(* CODESYS project BES3543.export

Project tree, tasks and I/O mapping:
  DATA_TYPE/
    data type EIXO_MOVER
    data type EIXO_STATUS
    data type RECEITA
    data type TURNOS_10
    function block COP [ST]
    function block FB_ATUADOR [ST]
    function block FB_Markem_SelecionarMacro [ST]
    function block FB_SMARTMOTOR [ST]
    program LEITURA_DATA_PLC [LD]
    function block RTON [FBD]
  D_PESAGEM/
    global variables GVL_PESAGEM
    program D00_PESAGEM [ST]
    program D01_EST_ETIQUETA [ST]
    program D02_SELEC_ETIQUETA [ST]
    program D03_ENTRADAS_REMOTAS [ST]
    program D04_SAIDAS_REMOTAS [ST]
  LADO_A/
    01 - LA_GERAL/
      global variables LA_GERAL
      program A00_ENTRADAS [ST]
      program A00_SAIDAS [ST]
      program A01_COMANDOS [ST]
      program A02_LAMPADAS [ST]
      program A03_COORDENADAS [ST]
      program ALARMES [ST]
    02 - LA_EMPILHADOR/
      global variables LA_EMP
      program B00_EMPILHA_SACOLA [ST]
      program B01_MANUAL [ST]
      program B02_EMPILHADOR_X [ST]
      program B03_INSPECAO [ST]
      program B04_ENTRADAS_REMOTAS [ST]
      program B05_SAIDAS_REMOTAS [ST]
    03 - LA_ENVOLVEDOR/
      global variables LA_ENV
      program C01_GIRO_SACOLA [ST]
      program C02_MANUAL [ST]
      program C03_EST_ENTRADA [ST]
      program C04_EST_TRANSPORTADOR [ST]
      program C05_EST_SAIDA [ST]
      program C06_ENTRADAS_REMOTAS [ST]
      program C07_SAIDAS_REMOTAS [ST]
    04 - LA_MOTION/
      program M0_LA_EMP_X [FBD]
      program M1_LA_EMP_GARRA [FBD]
      program M2_LA_EMP_GIRO [FBD]
      program M3_LA_ENV_Z [FBD]
      program M4_LA_ENV_X [FBD]
      program M5_LA_ENV_GIRO_LD [FBD]
      program M6_LA_ENV_GIRO_LE [FBD]
    05 - LA_IHM/
      global variables LA_IHM
      program E00_TELA_RECEITAS [ST]
      program E01_TELA_ATUADORES_EMPILHADOR [ST]
      program E02_TELA_ATUADORES_ENVOLVEDOR [ST]
      program E03_TELA_ATUADORES_PESAGEM [ST]
      program E04_TELA_OPERACAO [ST]
      program E05_CONTADORES [ST]
      program E06_HISTORICO [ST]
      program E07_HISTORICO_ESPELHAMENTO [ST]
  program TESTES_IOS [ST]
*)

// DATA_TYPE/EIXO_MOVER
TYPE EIXO_MOVER :
STRUCT
	
	sp_POSICAO			: LREAL;
	sp_VELOCIDADE		: LREAL;
	sp_ACELERACAO		: LREAL;
	sp_DESACELERACAO	: LREAL;

END_STRUCT
END_TYPE

// DATA_TYPE/EIXO_STATUS
TYPE EIXO_STATUS :
STRUCT
	
	bit_MOVE_FAZENDO		: BOOL;
	bit_MOVE_FEITO			: BOOL;
	bit_MOVE_ERRO			: BOOL;

END_STRUCT
END_TYPE

// DATA_TYPE/RECEITA
TYPE RECEITA :
STRUCT
	NOME 						: STRING;
	
	
//RECEITAS EMPILHADOR
	//CAMADAS MÁXIMAS DE EMPILHAMENTO / POSIÇÕES MÁXIMAS DE PEGA
	int_NUM_MAX_CAMADAS_EMPILHADOR	: INT;
	
	//CAMADA MÁXIMA DE EMPILHAMENTO ANTES DE ABAIXAR ATUADOR
	int_NUM_DESCER_MESA_EMPILHADOR	: INT;

	//GARRA EMPILHADOR
	coord_PRE_PEGA_GARRA_EMPILHADOR				: EIXO_MOVER;
	coord_PEGA_GARRA_EMPILHADOR					: EIXO_MOVER;
	
	sp_PRE_ENTREGA_GARRA_EMPILHADOR_POSICAO		: ARRAY[1..7] OF LREAL;
	sp_ENTREGA_GARRA_EMPILHADOR_VELOCIDADE		: LREAL;
	sp_ENTREGA_GARRA_EMPILHADOR_ACELERACAO		: LREAL;
	sp_ENTREGA_GARRA_EMPILHADOR_DESACELERACAO	: LREAL;
	
	sp_ENTREGA_GARRA_EMPILHADOR_POSICAO				: ARRAY[1..7] OF LREAL;
	sp_PRE_ENTREGA_GARRA_EMPILHADOR_VELOCIDADE		: LREAL;
	sp_PRE_ENTREGA_GARRA_EMPILHADOR_ACELERACAO		: LREAL;
	sp_PRE_ENTREGA_GARRA_EMPILHADOR_DESACELERACAO	: LREAL;
	
	tmr_TRANSICAO_ENTREGA_EMPILHADOR			: ARRAY[1..7] OF TIME;
	
	sp_POSICAO_ABRE_GARRA_EMPILHADOR			: ARRAY[1..7] OF LREAL;
	
	
	//EIXO X EMPILHADOR
	coord_X_EMPILHADOR_POS						: ARRAY[1..7] OF EIXO_MOVER;
	coord_X_EMPILHADOR_ENTREGA					: EIXO_MOVER;
	coord_X_EMPILHADOR_INSPECAO					: EIXO_MOVER;
	
	
	//MESA GIRO EMPILHADOR
	coord_MESA_GIRO_INICIAL				: EIXO_MOVER;
	coord_MESA_GIRO_FINAL				: EIXO_MOVER;
	coord_MESA_GIRO_INSPECAO			: EIXO_MOVER;
	
	
//RECEITAS ENVOLVEDOR
	//GIRO ENVOLVEDOR
	coord_GIRO_ENVOLVEDOR_PEGA			: EIXO_MOVER;
	coord_GIRO_ENVOLVEDOR_CORTE			: EIXO_MOVER;
	coord_GIRO_ENVOLVEDOR_ENTREGA		: EIXO_MOVER;
	
	//EIXO X ENVOLVEDOR
	coord_X_ENVOLVEDOR_PEGA				: EIXO_MOVER;
	coord_X_ENVOLVEDOR_CORTE			: EIXO_MOVER;
	coord_X_ENVOLVEDOR_ENTREGA			: EIXO_MOVER;
	
	//EIXO Z ENVOLVEDOR
	coord_Z_ENVOLVEDOR_PRE_PEGA			: EIXO_MOVER;
	coord_Z_ENVOLVEDOR_PEGA				: EIXO_MOVER;
	coord_Z_ENVOLVEDOR_SAIDA_PEGA		: EIXO_MOVER;
	coord_Z_ENVOLVEDOR_CORTE			: EIXO_MOVER;
	coord_Z_ENVOLVEDOR_ENTREGA			: EIXO_MOVER;
	
	int_NUMERO_GIROS_ENVOLVEDOR			: INT;
	
//PESO PILHA SACOLA
	num_PESO_SACOLA 				    : REAL;
			
END_STRUCT
END_TYPE

// DATA_TYPE/TURNOS_10
TYPE TURNOS_10 :
STRUCT
	PRIMEIRO		: ARRAY[0..9] OF DINT;
	SEGUNDO			: ARRAY[0..9] OF DINT;
	TERCEIRO		: ARRAY[0..9] OF DINT;
END_STRUCT
END_TYPE

// D_PESAGEM/GVL_PESAGEM
{attribute 'qualified_only'}
VAR_GLOBAL
	
	est_MESA_DE_TRANSFERENCIA				: BOOL;
	est_REJEITO_PRODUTO						: BOOL;
	est_TRANSPORTADOR_PESAGEM				: BOOL;
	est_TRANSPORTADOR_ESTAGIO_1				: BOOL;
	est_TRANNSPORTADOR_MERGER				: BOOL;
	
	est_MESA_DE_TRANSFERENCIA_REVERSE		: BOOL;
	est_TRANSPORTADOR_PESAGEM_REVERSE		: BOOL;
	
	
	bit_valv_ACIONAMENTO_TRANSFERENCIA		: BOOL;
	
	
	
	bit_PESANDO_PILHA_SACOLA				: BOOL;
	bit_ENVOLVEDOR_1						: BOOL;
	bit_ENVOLVEDOR_2						: BOOL;
	
	status_VALOR_PESAGEM					: WORD;
	array_ETIQUETA							: WORD;
	array_HIST_PESO							: WORD;
	
	
	bit_ENVOLVEDOR_ENVIANDO_PILHA_2			: BOOL;
	bit_PESAGEM_ATUAL						: BOOL;
	bit_PESAGEM_ERRO						: BOOL;
	bit_PESAGEM_OK							: BOOL;
	
	
//	ENTRADAS	============//============//============//============//============//============//============
	
	//E-16DIO - SLOT 5 (RMT50005)	
		di_SENS_MESA_TRANSFER_1				: BOOL;
		di_SENS_PRODUTO_BALANCA				: BOOL;
		di_BT_CMD1_INSPECAO_OK				: BOOL;
		di_feedback_ERRO_MESA_TRANSFER		: BOOL;
		di_feedback_ERRO_REJEITO_PRODUTO	: BOOL;
		di_SENS_MESA_TRANSFER_2				: BOOL;
		di_SENS_PRODUTO_REJEITO				: BOOL;
		di_SPEED_A_MERGER_1					: BOOL;
		
	//E-16DIO - SLOT 5 (RMT50006)	
		di_feedback_ERRO_ESTAGIO_1			: BOOL;
		di_SENS_TRANSFERENCIA_AV			: BOOL;
		di_SENS_ETIQUETADORA				: BOOL;
		di_SENS_POSICIONADOR_EMPILHADOR_RC	: BOOL;
		di_SENS_PRODUTO_DISPONIVEL			: BOOL;
		di_EST_MESA_TRANS_PESAGEM_DO1		: BOOL;
		di_SENS_TRANSFERENCIA_RC			: BOOL;
		di_SENS_PRODUTO_MERGER				: BOOL;
		di_SENS_POSICIONADOR_EMPILHADOR_AV	: BOOL;
		di_feedback_ERRO_MERGER_1			: BOOL;;
		
	
//	SAIDAS		============//============//============//============//============//============//============

	//E-16DIO - SLOT 5 (RMT50005)
		do_SPEED_A_MESA_TRANSFER		: BOOL;
		do_ATU_TRANSFERENCIA_RC			: BOOL;
		do_LAMP_INSPECAO_OK				: BOOL;
		do_REVERSE_MESA_TRANSFER		: BOOL;
		do_SPEED_B_MESA_TRANSFER		: BOOL;
		do_SPEED_A_REJEITO_PRODUTO		: BOOL;
		do_ATU_TRANSFERENCIA_AV			: BOOL;
		
	//E-16DIO - SLOT 6 (RMT50006)
		do_EST_MESA_TRANS_PESAGEM_DI2	: BOOL;
		do_EST_MESA_TRANS_PESAGEM_DI3	: BOOL;
		do_ATU_POSICIONADOR_RC			: BOOL;
		do_EST_MESA_TRANS_PESAGEM_DI1	: BOOL;
		do_SPEED_A_ESTAGIO_1			: BOOL;
		do_ATU_POSICIONADOR_AV			: BOOL;
		
	//E-16DIO - SLOT 7 (RMT50007)
		do_EST_BALANCA					: BOOL;
		do_est_BALANCA_REVERSE			: BOOL;
	
END_VAR

// LADO_A/01 - LA_GERAL/LA_GERAL
{attribute 'qualified_only'}
VAR_GLOBAL

//Teste teste teste	
//RECEITAS
	rec_IHM								: RECEITA;
	rec_SELECIONADA						: RECEITA;

//COMANDOS
	bit_MAQUINA_PRONTA				: BOOL;
	bit_MAQUINA_RODANDO				: BOOL;
	bit_MAQUINA_RESET				: BOOL;
	bit_MAQUINA_ESTAVEL				: BOOL;
	bit_SERVOS_RESET				: BOOL;
	bit_SAFETY_ATIVO				: BOOL;
	
	bit_MAQUINA_MANUAL				: BOOL;
	bit_BT_DESLIGA					: BOOL;
	
	
	bit_SERVOS_ENABLE				: BOOL;
	bit_AUTO_HABILITAR_EIXOS		: BOOL;
	bit_EIXO_X_EMPILHADOR_PRONTO	: BOOL;
	bit_EIXO_GARRA_EMPILHADOR_PRONTO : BOOL;
	bit_EIXO_GIRO_MESA_PRONTO		: BOOL;
	bit_EIXO_Z_ENVOLVEDOR_PRONTO	: BOOL;
	bit_EIXO_X_ENVOLVEDOR_PRONTO	: BOOL;
	bit_EIXO_GIRO_ENVOLVEDOR_LD_PRONTO : BOOL;
	bit_EIXO_GIRO_ENVOLVEDOR_LE_PRONTO : BOOL;
	bit_EIXOS_PRONTOS				: BOOL;
	
	TESTE_Z							: BOOL;
	RESET_Z							: BOOL;
	bit_TIRANDO_PRODUTO				: BOOL;
	bit_ALARME_SONORO_CASE			: BOOL;
	bit_SACOLA_POSICIONADA				: BOOL;
	tmr_CICLO_COMPLETO				: TON;

//LAMPADAS
	bit_LAMP_VERDE					: BOOL;
	bit_LAMP_VERMELHO				: BOOL;
	bit_LAMP_AMARELO				: BOOL;
	bit_LAMP_AZUL					: BOOL;
	bit_TL_SONORO					: BOOL;
	bit_LAMP_INSPECAO				: BOOL;
		
	bit_LAMP_VERDE_PULSO			: BOOL;
	bit_LAMP_VERMELHO_PULSO			: BOOL;
	bit_LAMP_AMARELO_PULSO			: BOOL;
	bit_LAMP_AZUL_PULSO				: BOOL;
	bit_TL_SONORO_PULSO				: BOOL;
	bit_LAMP_INSPECAO_PULSO			: BOOL;
	
//ALARMES
	status_alarm_EIXO_Y					: INT;
	status_alarm_EIXO_Z					: INT;
	status_alarm_EIXO_COLMEIA_1			: INT;
	status_alarm_EIXO_COLMEIA_2			: INT;
	status_alarm_atu_POSICIONA_PRODUTO	: INT;
	status_alarm_atu_STOP_ENTREGA		: INT;
	status_alarm_atu_STOP_PRE_ENTREGA	: INT;
	status_alarm_atu_MANI_GARRA			: INT;
	status_alarm_atu_PRODUTO_FREIO		: INT;
	status_alarm_atu_SEPARADOR_Y		: INT;
	status_alarm_atu_SEPARADOR_Z		: INT;
	status_alarm_atu_DIVERTER_FREIO		: INT;
	
	status_alarm_atu_FORM_PEGA_CAIXA	: INT;
	status_alarm_atu_FORM_FORMADOR		: INT;
	status_alarm_atu_FORM_EMPURADDOR	: INT;
	status_alarm_atu_FORM_VACUO			: INT;
	
	status_alarm_SAFETY_CASE			: INT;
	status_alarm_SAFETY_FORM			: INT;
	status_alarm_AR						: INT;
	
	status_alarm_in_PORTA_CASE_1		: INT;
	status_alarm_in_PORTA_CASE_2		: INT;
	status_alarm_in_PORTA_CASE_3		: INT;
	status_alarm_in_PORTA_CASE_4		: INT;
	status_alarm_in_PORTA_CASE_5		: INT;
	
	bit_STATUS_PARADA					: BOOL;
	bit_STATUS_OCIOSA					: BOOL;
	bit_STATUS_RODANDO					: BOOL;
	
	bit_TURNO_TROCADO					: BOOL;
	
	status_alarm_HOME_EIXO_Y			: INT;
	status_alarm_HOME_EIXO_Z			: INT;
	status_alarm_HOME_DIVERTER			: INT;
	status_alarm_ACUMULO_CAIXAS			: INT;
	status_alarm_in_PORTA_DIVERTER		: INT;
	status_alarm_VACUO_COLMEIA			: INT;
	status_alarm_NIVEL_COLMEIA			: INT;
	status_alarm_VACUO_PRODUTOS			: INT;
	status_alarm_INDEX_CAIXAS			: INT;
	status_alarm_COLMEIA_FREIO			: INT;
	status_alarm_BRACO_COLMEIA			: INT;
	status_alarm_FALTA_CAIXA			: INT;
	status_alarm_FALHA_PEGA				: INT;
	status_alarm_TEMP_COLA				: INT;
	status_alarm_NIVEL_COLA				: INT;
	status_alarm_BT_EMERGENCIA_CASE_1	: INT;
	status_alarm_BT_EMERGENCIA_CASE_2	: INT;
	status_alarm_BT_EMERGENCIA_FORM		: INT;
	atu_DESVIO_RODA						: BOOL;
	
	bit_ALARME_AR_CASE_ATIVO			: BOOL;
	bit_ALARME_FALTA_CAIXA_ATIVO		: BOOL;
	bit_SONORO_PULSO					: BOOL;
	
	r_trig_SEM_COLMEIA					: R_TRIG;
	r_trig_COLMEIA						: R_TRIG;
	bit_HABILITAR_EIXOS					: BOOL;
	
//	COORDENADAS	============//============//============//============//============//============//============
	
	//GARRA EMPILHADOR
	coord_GARRA_EMPILHADOR_PRE_PEGA						: EIXO_MOVER;
	coord_GARRA_EMPILHADOR_PEGA							: EIXO_MOVER;
	coord_GARRA_EMPILHADOR_PRE_ENTREGA					: EIXO_MOVER;
	coord_GARRA_EMPILHADOR_ENTREGA						: EIXO_MOVER;
	
	//EIXO X EMPILHADOR
	coord_X_EMPILHADOR_POS_1							: EIXO_MOVER;
	coord_X_EMPILHADOR_POS_2							: EIXO_MOVER;
	coord_X_EMPILHADOR_POS_3							: EIXO_MOVER;
	coord_X_EMPILHADOR_POS_4							: EIXO_MOVER;
	coord_X_EMPILHADOR_POS_5							: EIXO_MOVER;
	coord_X_EMPILHADOR_POS_6							: EIXO_MOVER;
	
	coord_X_EMPILHADOR_INSPECAO							: EIXO_MOVER;
	coord_X_EMPILHADOR_ENTREGA							: EIXO_MOVER;
	
	//MESA GIRO EMPILHADOR
	coord_MESA_GIRO_POSICAO_INICIAL						: EIXO_MOVER;
	coord_MESA_GIRO_POSICAO_FINAL						: EIXO_MOVER;
	coord_MESA_GIRO_POSICAO_INSPECAO					: EIXO_MOVER;
	
	
	//EIXO Z ENVOLVEDOR
	coord_Z_ENVOLVEDOR_PRE_PEGA							: EIXO_MOVER;
	coord_Z_ENVOLVEDOR_PEGA								: EIXO_MOVER;
	coord_Z_ENVOLVEDOR_SAIDA_PEGA						: EIXO_MOVER;
	coord_Z_ENVOLVEDOR_CORTE							: EIXO_MOVER;
	coord_Z_ENVOLVEDOR_ENTREGA							: EIXO_MOVER;
	
	
	//EIXO X ENVOLVEDOR
	coord_X_ENVOLVEDOR_PEGA								: EIXO_MOVER;
	coord_X_ENVOLVEDOR_CORTE							: EIXO_MOVER;
	coord_X_ENVOLVEDOR_ENTREGA							: EIXO_MOVER;
	
	
	//GIRO ENVOLVEDOR
	coord_GIRO_ENVOLVEDOR_PEGA							: EIXO_MOVER;
	coord_GIRO_ENVOLVEDOR_CORTE							: EIXO_MOVER;
	coord_GIRO_ENVOLVEDOR_ENTREGA						: EIXO_MOVER;
	
	
//	ENTRADAS	============//============//============//============//============//============//============

	//E-16DI - SLOT 1
		di_BT_CMD1_START				: BOOL;
		di_BT_CMD1_STOP					: BOOL;
		di_BT_CMD1_RESET				: BOOL;
		di_BT_CMD2_START				: BOOL;
		di_BT_CMD2_STOP					: BOOL;
		di_BT_CMD2_RESET				: BOOL;
		di_SEG_GERAL_ATIVA				: BOOL;
		di_SEG_INTERNA_ATIVA			: BOOL;
		di_SEG_PORTA_1					: BOOL;
		di_SEG_PORTA_2					: BOOL;
		
	//E-16DI - SLOT 2
		di_ENV_SENS_ATU_GARRA_LD_RC		: BOOL;
		di_ENV_SENS_ATU_GARRA_LE_RC		: BOOL;
		di_ENV_SENS_ATU_ABERTURA_AV		: BOOL;
		di_ENV_SENS_ATU_ABERTURA_RC		: BOOL;
	
//	SAIDAS		============//============//============//============//============//============//============

	//E-8DO - SLOT 3
		do_TL1_VERDE				: BOOL;
		do_TL1_VERMELHO				: BOOL;
		do_TL1_AMARELO				: BOOL;
		do_TL2_VERDE				: BOOL;
		do_TL2_VERMELHO				: BOOL;
		do_TL2_AMARELO				: BOOL;
		do_TL1_SONORO				: BOOL;
		do_SAIDA_COLAR_EQUIQUETA	: BOOL;
		
	//E-8DO - SLOT 4
		do_ENV_CORTE_FILME			: BOOL;
		
	//E-8DO - SLOT 5
		do_ENV_ATU_GARRAS			: BOOL;
		do_ENV_ATU_ABERTURA			: BOOL;	

	
	bit_MAQUINA_VAZIO					: BOOL;
	
	int_HIST_INDEX_TURNO1			: DINT;
	int_HIST_INDEX_TURNO2			: DINT;
	int_HIST_INDEX_TURNO3			: DINT;
	
	num_VOLTAS							: LREAL;
	
	bit_EIXO_GERAL_MOVENDO			: BOOL;
	
	bit_RESET_GERAL					: BOOL;
	
END_VAR

// LADO_A/02 - LA_EMPILHADOR/LA_EMP
{attribute 'qualified_only'}
VAR_GLOBAL
	
//COMANDOS

	bit_GARRA_EMPILHADOR_EXECUTANDO_RESET	: BOOL;
	bit_EIXO_X_EMPILHADOR_EXECUTANDO_RESET	: BOOL;
	bit_MESA_GIRO_EXECUTANDO_RESET			: BOOL;
	
	bit_ENTREGA_EMPILHADOR_CONCLUIDO		: BOOL;
	bit_ENTREGA_PILHA_CONCLUIDO				: BOOL;
	bit_EIXO_X_MOVE_CONCLUIDO				: BOOL;
	bit_MESA_GIRO_CONCLUIDO					: BOOL;
	
	bit_LIBERA_INSPECAO_PILHA				: BOOL;
	bit_EST_INSPECAO_ENTREGUE_1				: BOOL;
	bit_EST_INSPECAO_ENTREGUE_2				: BOOL;
	bit_OPERADOR_INSPECAO_OK				: BOOL;
	bit_EST_ENVIAR_PILHA_INSPECAO			: BOOL;
	bit_REALIZANDO_INSPECAO					: BOOL;
	
	bit_LIBERA_ENTREGA_PILHA				: BOOL;
	bit_ENTREGANDO_PILHA_COMPLETA			: BOOL;
	bit_EST_PILHA_ENTREGUE					: BOOL;
	
	bit_STATUS_INSPECAO_1					: BOOL;
	
	bit_LIBERA_PEGA							: BOOL;
	bit_LIBERA_GIRO							: BOOL;
	bit_LIBERA_X							: BOOL;
	
	bit_PILHA_PAR							: BOOL;
	bit_PILHA_IMPAR							: BOOL;
	
	bit_GIRO_MESA_REVERSE					: BOOL;
	bit_GIRO_MESA_FOWARD					: BOOL;
	
	bit_LIGA_EST_INSPECAO					: BOOL;
	bit_LIGA_EST_MESA_GIRO					: BOOL;
	
	
	bit_valv_GARRA_SACOLA					: BOOL;
	bit_valv_BANDEJA						: BOOL;
	bit_valv_DESCE_MESA_GIRO				: BOOL;
	bit_valv_POSICIONA_SACOLA				: BOOL;
	
	est_ROLETES_GIRO_MESA					: BOOL;
	est_INSPECAO_EMPILHADOR 				: BOOL;
	
	est_ROLETES_GIRO_MESA_REVERSE			: BOOL;
	est_INSPECAO_EMPILHADOR_REVERSE			: BOOL;
	
	
	
	
	bit_EIXO_X_EMPILHADOR_FAZER_HOME		: BOOL;
	bit_EIXO_X_EMPILHADOR_POSICIONADO		: BOOL;
	
	bit_EIXO_GIRO_MESA_FAZER_HOME			: BOOL;
	bit_EIXO_GIRO_MESA_POSICIONADO			: BOOL;
	
	bit_EIXO_GARRA_EMPILHADOR_FAZER_HOME	: BOOL;
	bit_EIXO_GARRA_EMPILHADOR_POSICIONADO	: BOOL;
	
	
	
	bit_EIXO_GARRA_EMPILHADOR_MOVER_ABS		: BOOL;
	bit_EIXO_GARRA_EMPILHADOR_MOVER_REL		: BOOL;
	
	bit_EIXO_X_EMPILHADOR_MOVER_ABS			: BOOL;
	bit_EIXO_X_EMPILHADOR_MOVER_REL			: BOOL;
	
	bit_EIXO_GIRO_MESA_MOVER_ABS			: BOOL;
	bit_EIXO_GIRO_MESA_MOVER_REL			: BOOL;
	

	
	bit_GARRA_EMPILHADOR_JOG_FORWARD		: BOOL;
	bit_GARRA_EMPILHADOR_JOG_REVERSE		: BOOL;
	bit_GARRA_EMPILHADOR_JOG_STOP			: BOOL;
	
	bit_EIXO_X_EMPILHADOR_JOG_FORWARD		: BOOL;
	bit_EIXO_X_EMPILHADOR_JOG_REVERSE		: BOOL;
	bit_EIXO_X_EMPILHADOR_JOG_STOP			: BOOL;
	
	bit_GIRO_MESA_JOG_FORWARD				: BOOL;
	bit_GIRO_MESA_JOG_REVERSE				: BOOL;
	bit_GIRO_MESA_JOG_STOP					: BOOL;
	
	
	info_MOTOR_GARRA_EMPILHADOR_POS_ATUAL	: LREAL;
	info_MOTOR_EIXO_X_EMPILHADOR_POS_ATUAL	: LREAL;
	info_MOTOR_GIRO_MESA_POS_ATUAL			: LREAL;
	
	
	num_GIROS_STRETCH					: LREAL;
	
	tmr_RTON_MOVE_1						: RTON;
	tmr_RTON_MOVE_2						: RTON;
	tmr_RTON_MOVE_3						: RTON;
	tmr_RTON_MOVE_4						: RTON;
	tmr_RTON_MOVE_5						: RTON;
	
	
	//	ENTRADAS	============//============//============//============//============//============//============
		
	//E-16DIO - SLOT 1 (RMT50001)	
		di_SENS_MESA_GIRO_RC				: BOOL;
		di_SENS_MESA_GIRO_MD				: BOOL;
		di_SENS_PINCA_GARRA_EMPILHADOR_RC	: BOOL;
		di_SENS_APOIO_BANDEJA_RC			: BOOL;
		di_SENS_EST_INSPEC_PRODUTO_1		: BOOL;
		di_SENS_MESA_GIRO_AV				: BOOL;
		di_SENS_PINCA_GARRA_EMPILHADOR_AV	: BOOL;
		di_SENS_APOIO_BANDEJA_AV			: BOOL;
		di_SENS_PRODUTO_MESA_GIRO			: BOOL;
		di_SENS_EST_INSPEC_PRODUTO_2		: BOOL;
		
	//E-16DIO - SLOT 2 (RMT50002)	
		di_feedback_ERRO_MESA_GIRO			: BOOL;
		di_feedback_ERRO_EST_INSPECAO		: BOOL;
		
	
	
//	SAIDAS		============//============//============//============//============//============//============

	//E-16DIO - SLOT 1 (RMT50001)		
		do_ATU_MESA_GIRO_RC				: BOOL;
		do_ATU_PINCA_GARRA_EMPILHADOR	: BOOL;
		do_ATU_MESA_GIRO_AV				: BOOL;
		do_ATU_BANDEJA_APOIO			: BOOL;
		
	//E-16DIO - SLOT 2 (RMT50002)	
		do_SPEED_A_MESA_GIRO			: BOOL;
		do_SPEED_A_EST_INSPECAO			: BOOL;
		do_REVERSE_MESA_GIRO			: BOOL;
		do_SPEED_B_MESA_GIRO			: BOOL;
		do_REVERSE_EST_INSPECAO			: BOOL;
		do_SPEED_B_EST_INSPECAO			: BOOL;
		
	
	
	
	
END_VAR

// LADO_A/03 - LA_ENVOLVEDOR/LA_ENV
{attribute 'qualified_only'}
VAR_GLOBAL

	//BITS DE COMANDOS
	bit_ENVOLVEDOR_SACOLA_POSICIONADA		: BOOL;
	bit_ENVOLVEDOR_SACOLA_DEPOSITANDO		: BOOL;
	bit_ENVOLVEDOR_SACOLA_DEPOSITADA		: BOOL;
	
	bit_ENVOLVEDOR_ENVIANDO_PILHA			: BOOL;
	
	
	bit_EST_ENTRADA_CHEIA					: BOOL;

	

	//ATUADORES
	bit_valv_APROX_GARRA			: BOOL;
	bit_valv_GARRA_DUPLA			: BOOL;
	bit_valv_CORTE_FILME			: BOOL;
	bit_valv_VACUO_FILME			: BOOL;
	bit_ENV_CORTE_FILME			: BOOL;
	bit_valv_FECHA_FILME_1			: BOOL;
	bit_valv_FECHA_FILME_2			: BOOL;
	bit_valv_FECHA_FILME_3			: BOOL;
	
	//ESTEIRAS
	est_ENTRADA_ENVOLVEDOR			: BOOL;
	est_TRANSPORTADOR_ENVOLVEDOR	: BOOL;
	est_SAIDA_ENVOLVEDOR			: BOOL;


	//BITS DE EIXOS
	bit_EIXO_Z_ENVOLVEDOR_FAZER_HOME			: BOOL;
	bit_EIXO_Z_ENVOLVEDOR_POSICIONADO			: BOOL;
	
	bit_EIXO_X_ENVOLVEDOR_FAZER_HOME			: BOOL;
	bit_EIXO_X_ENVOLVEDOR_POSICIONADO			: BOOL;

	bit_EIXO_GIRO_ENVOLVEDOR_LD_FAZER_HOME		: BOOL;
	bit_EIXO_GIRO_ENVOLVEDOR_LD_POSICIONADO		: BOOL;
	
	bit_EIXO_GIRO_ENVOLVEDOR_LE_FAZER_HOME		: BOOL;
	bit_EIXO_GIRO_ENVOLVEDOR_LE_POSICIONADO		: BOOL;
	
	
	
	bit_EIXO_Z_ENVOLVEDOR_MOVER_ABS				: BOOL;
	bit_EIXO_Z_ENVOLVEDOR_MOVER_REL				: BOOL;
	
	bit_EIXO_X_ENVOLVEDOR_MOVER_ABS				: BOOL;
	bit_EIXO_X_ENVOLVEDOR_MOVER_REL				: BOOL;
	
	bit_EIXO_GIRO_ENVOLVEDOR_LD_MOVER_ABS		: BOOL;
	bit_EIXO_GIRO_ENVOLVEDOR_LD_MOVER_REL		: BOOL;
	
	bit_EIXO_GIRO_ENVOLVEDOR_LE_MOVER_ABS		: BOOL;
	bit_EIXO_GIRO_ENVOLVEDOR_LE_MOVER_REL		: BOOL;
	
	
	bit_MOTOR_Z_ENVOLVEDOR_JOG_FORWARD			: BOOL;
	bit_MOTOR_Z_ENVOLVEDOR_JOG_REVERSE			: BOOL;
	bit_MOTOR_Z_ENVOLVEDOR_JOG_STOP				: BOOL;
	
	bit_MOTOR_X_ENVOLVEDOR_JOG_FORWARD			: BOOL;
	bit_MOTOR_X_ENVOLVEDOR_JOG_REVERSE			: BOOL;
	bit_MOTOR_X_ENVOLVEDOR_JOG_STOP				: BOOL;
	
	bit_MOTOR_GIRO_ENVOLVEDOR_LD_JOG_FORWARD	: BOOL;
	bit_MOTOR_GIRO_ENVOLVEDOR_LD_JOG_REVERSE	: BOOL;
	bit_MOTOR_GIRO_ENVOLVEDOR_LD_JOG_STOP		: BOOL;
	
	bit_MOTOR_GIRO_ENVOLVEDOR_LE_JOG_FORWARD	: BOOL;
	bit_MOTOR_GIRO_ENVOLVEDOR_LE_JOG_REVERSE	: BOOL;
	bit_MOTOR_GIRO_ENVOLVEDOR_LE_JOG_STOP		: BOOL;
	
	info_MOTOR_GIRO_ENVOLVIMENTO_LD_POS_ATUAL	: LREAL;
	info_MOTOR_GIRO_ENVOLVIMENTO_LE_POS_ATUAL	: LREAL;
	
	info_MOTOR_Z_ENVOLVEDOR_POS_ATUAL			: LREAL;
	info_MOTOR_X_ENVOLVEDOR_POS_ATUAL			: LREAL;

	
	
//	ENTRADAS	============//============//============//============//============//============//============

	
	//E-16DIO - SLOT 3 (RMT50003)	
		di_SENS_EST_TRANS_PRESENCA			: BOOL;
		di_SENS_POS_2_ENVOLVEDOR			: BOOL;
		di_SENS_CORTE_FILME_RC				: BOOL;
		di_feedback_ERRO_ENTRADA_ENVOLVEDOR : BOOL;
		di_SENS_POS_1_ENVOLVEDOR			: BOOL;
		di_SENS_FILME_ENVOLVEDOR			: BOOL;
		di_SENS_CORTE_FILME_AV				: BOOL;
	
	//E-16DIO - SLOT 4 (RMT50004)		
		di_SENS_SAIDA_ENVOLVEDOR_1			: BOOL;
		di_SENS_SAIDA_ENVOLVEDOR_3			: BOOL;
		di_SENS_FECHA_FILME_1_RC			: BOOL;
		di_SENS_FECHA_FILME_2_RC			: BOOL;
		di_SENS_FECHA_FILME_3_RC			: BOOL;
		di_feedback_ERRO_TRANSP_SAIDA_1		: BOOL;
		di_SENS_SAIDA_ENVOLVEDOR_2			: BOOL;
		di_SENS_SAIDA_ENVOLVEDOR_4			: BOOL;
		di_SENS_FECHA_FILME_2_AV			: BOOL;
		di_SENS_FECHA_FILME_3_AV			: BOOL;

		
		
//	SAIDAS		============//============//============//============//============//============//============

	//E-16DIO - SLOT 3 (RMT50003)	
		do_EST_TRANS_ENVOLVEDOR_DI2		: BOOL;
		do_EST_TRANS_ENVOLVEDOR_DI3		: BOOL;
		do_VALV_CORTE_FILME				: BOOL;
		do_SPEED_A_ENTRADA_ENVOLVEDOR	: BOOL;
		do_EST_TRANS_ENVOLVEDOR_DI1		: BOOL;
		do_EST_TRANS_ENVOLVEDOR_DO1		: BOOL;
		do_VALV_VACUO_FILME				: BOOL;
		
	//E-16DIO - SLOT 4 (RMT50004)
		do_VALV_FECHA_FILME_2			: BOOL;
		do_SPEED_A_TRANSP_SAIDA_1		: BOOL;
		do_VALV_FECHA_FILME_1			: BOOL;
		do_VALV_FECHA_FILME_3			: BOOL;
	
	
END_VAR

// LADO_A/05 - LA_IHM/LA_IHM
{attribute 'qualified_only'}
VAR_GLOBAL
	
//Tela de Operação
	bit_MAQUINA_MANUAL				: BOOL;
	bit_MANUAL_HABILITAR_EIXOS		: BOOL;
	bit_bt_INSPECAO_OK				: BOOL;
	bit_STATUS_INSPECAO_OK			: INT;
	bit_STATUS_PESAGEM				: INT;
	
	
	array_HIST_ERRO_PESAGEM_1		: BOOL;
	array_HIST_ERRO_PESAGEM_2		: BOOL;
	array_HIST_ERRO_PESAGEM_3		: BOOL;
	array_HIST_ERRO_PESAGEM_4		: BOOL;
	array_HIST_ERRO_PESAGEM_5		: BOOL;
	array_HIST_ERRO_PESAGEM_6		: BOOL;
	array_HIST_ERRO_PESAGEM_7		: BOOL;


//ICONES DE ALARME NOS EIXOS
	bit_EIXO_X_EMPILHADOR_ALARME_ATIVO			: BOOL;
	bit_EIXO_GARRA_EMPILHADOR_ALARME_ATIVO		: BOOL;
	bit_EIXO_GIRO_MESA_ALARME_ATIVO				: BOOL;
	bit_EIXO_Z_ENVOLVEDOR_ALARME_ATIVO			: BOOL;
	bit_EIXO_X_ENVOLVEDOR_ALARME_ATIVO			: BOOL;
	bit_EIXO_GIRO_ENVOLVEDOR_LD_ALARME_ATIVO	: BOOL;
	bit_EIXO_GIRO_ENVOLVEDOR_LE_ALARME_ATIVO	: BOOL;
	bit_EIXO_GERAL_SAFETY						: BOOL;

//ICONES DE EIXOS HABILITADOS	
	bit_EIXO_X_EMPILHADOR_HABILITADO			: BOOL;
	bit_EIXO_GARRA_EMPILHADOR_HABILITADO		: BOOL;
	bit_EIXO_GIRO_MESA_HABILITADO				: BOOL;
	bit_EIXO_Z_ENVOLVEDOR_HABILITADO			: BOOL;
	bit_EIXO_X_ENVOLVEDOR_HABILITADO			: BOOL;
	bit_EIXO_GIRO_ENVOLVEDOR_LD_HABILITADO		: BOOL;
	bit_EIXO_GIRO_ENVOLVEDOR_LE_HABILITADO		: BOOL;
	
//ICONES PARA MOVIMENTOS JOG DOS EIXOS	
	bit_EIXO_X_EMPILHADOR_JOG_POSITIVO			: BOOL;
	bit_EIXO_X_EMPILHADOR_JOG_NEGATIVO			: BOOL;
	bit_EIXO_GARRA_EMPILHADOR_JOG_POSITIVO		: BOOL;
	bit_EIXO_GARRA_EMPILHADOR_JOG_NEGATIVO		: BOOL;
	bit_EIXO_GIRO_MESA_JOG_POSITIVO				: BOOL;
	bit_EIXO_GIRO_MESA_JOG_NEGATIVO				: BOOL;
	bit_EIXO_Z_ENVOLVEDOR_JOG_POSITIVO			: BOOL;
	bit_EIXO_Z_ENVOLVEDOR_JOG_NEGATIVO			: BOOL;
	bit_EIXO_X_ENVOLVEDOR_JOG_POSITIVO			: BOOL;
	bit_EIXO_X_ENVOLVEDOR_JOG_NEGATIVO			: BOOL;
	bit_EIXO_GIRO_ENVOLVEDOR_LD_JOG_POSITIVO	: BOOL;
	bit_EIXO_GIRO_ENVOLVEDOR_LD_JOG_NEGATIVO	: BOOL;
	bit_EIXO_GIRO_ENVOLVEDOR_LE_JOG_POSITIVO	: BOOL;
	bit_EIXO_GIRO_ENVOLVEDOR_LE_JOG_NEGATIVO	: BOOL;
	
//ICONES PARA FAZER HOME DOS EIXOS	
	bit_EIXO_X_EMPILHADOR_FAZER_HOME			: BOOL;
	bit_EIXO_GARRA_EMPILHADOR_FAZER_HOME		: BOOL;
	bit_EIXO_GIRO_MESA_FAZER_HOME				: BOOL;
	bit_EIXO_Z_ENVOLVEDOR_FAZER_HOME			: BOOL;
	bit_EIXO_X_ENVOLVEDOR_FAZER_HOME			: BOOL;
	bit_EIXO_GIRO_ENVOLVEDOR_LD_FAZER_HOME		: BOOL;
	bit_EIXO_GIRO_ENVOLVEDOR_LE_FAZER_HOME		: BOOL;
	
	
	//ICONES DE STATUS DO HOME DOS EIXOS
	bit_EIXO_X_EMPILHADOR_FAZENDO_HOME			: BOOL;
	bit_EIXO_GARRA_EMPILHADOR_FAZENDO_HOME		: BOOL;
	bit_EIXO_GIRO_MESA_FAZENDO_HOME				: BOOL;
	bit_EIXO_Z_ENVOLVEDOR_FAZENDO_HOME			: BOOL;
	bit_EIXO_X_ENVOLVEDOR_FAZENDO_HOME			: BOOL;
	bit_EIXO_GIRO_ENVOLVEDOR_LD_FAZENDO_HOME	: BOOL;
	bit_EIXO_GIRO_ENVOLVEDOR_LE_FAZENDO_HOME	: BOOL;
	
		
//INFORMAÇÃO DE POSIÇÃO ATUAL
	info_MANI_POS_ATUAL_X_EMPILHADOR			: LREAL;
	info_MANI_POS_ATUAL_GIRO_MESA				: LREAL;
	info_MANI_POS_ATUAL_Z_ENVOLVEDOR			: LREAL;
	info_MANI_POS_ATUAL_X_ENVOLVEDOR			: LREAL;
	info_MANI_POS_ATUAL_GARRA_EMPILHADOR		: LREAL;
	info_POS_ATUAL_GIRO_EMPILHADOR_LD			: LREAL;
	info_POS_ATUAL_GIRO_EMPILHADOR_LE			: LREAL;
	
	
//ICONES DE ALARME NOS MOTORES
	bit_feedback_ERRO_MESA_GIRO				: BOOL;
	bit_feedback_ERRO_EST_INSPECAO			: BOOL;
	bit_feedback_ERRO_ENTRADA_ENVOLVEDOR	: BOOL;
	bit_feedback_ERRO_TRANSP_SAIDA_1		: BOOL;
	bit_feedback_ERRO_MESA_TRANSFER			: BOOL;
	bit_feedback_ERRO_REJEITO_PRODUTO		: BOOL;
	bit_feedback_ERRO_ESTAGIO_1				: BOOL;
	bit_feedback_ERRO_MERGER_1				: BOOL;
	
	
	
	bit_GIRO_SACOLA_RESET			: BOOL;
	bit_GIRO_EMPILHAMENTO_RESET		: BOOL;
	
	sp_MANI_VELOCIDADE				: UINT;
	
	int_CAMADA_ATUAL				: INT	:=	1;
	
	bit_SIMULA_PEGA					: BOOL;
	bit_SIMULA_GIRO					: BOOL;
	bit_bt_RESET_SERVO				: BOOL;

// Tela de Receita
	bt_CARREGAR_RECEITA				: BOOL;
	bt_SALVAR_RECEITA				: BOOL;
	bt_UPLOAD_RECEITA				: BOOL;
	bt_DOWNLOAD_RECEITA				: BOOL;
	
	int_RECEITA_ATUAL				: INT;
	int_STATUS_RECEITA				: INT;
	
	
	bit_SELEC_RECEITA_1				: BOOL;
	bit_SELEC_RECEITA_2				: BOOL;
	bit_SELEC_RECEITA_3				: BOOL;
	bit_SELEC_RECEITA_4				: BOOL;
	bit_SELEC_RECEITA_5				: BOOL;
	bit_SELEC_RECEITA_6				: BOOL;
	bit_SELEC_RECEITA_7				: BOOL;
	bit_SELEC_RECEITA_8				: BOOL;
	bit_SELEC_RECEITA_9				: BOOL;
	bit_SELEC_RECEITA_10			: BOOL;
	
	
	nome_RECEITA_1							: STRING;
	nome_RECEITA_2							: STRING;
	nome_RECEITA_3							: STRING;
	nome_RECEITA_4							: STRING;
	nome_RECEITA_5							: STRING;
	nome_RECEITA_6							: STRING;
	nome_RECEITA_7							: STRING;
	nome_RECEITA_8							: STRING;
	nome_RECEITA_9							: STRING;
	nome_RECEITA_10							: STRING;
	
	
	ALARME_ATIVO					: BOOL;
	
	TEMPO_1				: TIME;
	TEMPO_2				: TIME;
	TEMPO_3				: TIME;
	TEMPO_4				: TIME;
	TEMPO_5				: TIME;
	TEMPO_TOTAL			: TIME;
	TEMPO_TOTAL_2		: TIME;
	
	bit_RESET_RTON		: BOOL;
	
//CONTADORES DE TEMPO DE MAQUINA
	//TURNO 1
	num_MAQUINA_RODANDO_SEGUNDOS_T1	: DINT;
	num_MAQUINA_RODANDO_MINUTOS_T1	: DINT;
	num_MAQUINA_RODANDO_HORAS_T1	: DINT;
	
	num_MAQUINA_PARADA_SEGUNDOS_T1	: DINT;
	num_MAQUINA_PARADA_MINUTOS_T1	: DINT;
	num_MAQUINA_PARADA_HORAS_T1		: DINT;
	
	num_MAQUINA_OCIOSA_SEGUNDOS_T1	: DINT;
	num_MAQUINA_OCIOSA_MINUTOS_T1	: DINT;
	num_MAQUINA_OCIOSA_HORAS_T1		: DINT;
	
	
	//TURNO 2
	num_MAQUINA_RODANDO_SEGUNDOS_T2	: DINT;
	num_MAQUINA_RODANDO_MINUTOS_T2	: DINT;
	num_MAQUINA_RODANDO_HORAS_T2	: DINT;
	
	num_MAQUINA_PARADA_SEGUNDOS_T2	: DINT;
	num_MAQUINA_PARADA_MINUTOS_T2	: DINT;
	num_MAQUINA_PARADA_HORAS_T2		: DINT;
	
	num_MAQUINA_OCIOSA_SEGUNDOS_T2	: DINT;
	num_MAQUINA_OCIOSA_MINUTOS_T2	: DINT;
	num_MAQUINA_OCIOSA_HORAS_T2		: DINT;
	
	
	//TURNO 3
	num_MAQUINA_RODANDO_SEGUNDOS_T3	: DINT;
	num_MAQUINA_RODANDO_MINUTOS_T3	: DINT;
	num_MAQUINA_RODANDO_HORAS_T3	: DINT;
	
	num_MAQUINA_PARADA_SEGUNDOS_T3	: DINT;
	num_MAQUINA_PARADA_MINUTOS_T3	: DINT;
	num_MAQUINA_PARADA_HORAS_T3		: DINT;
	
	num_MAQUINA_OCIOSA_SEGUNDOS_T3	: DINT;
	num_MAQUINA_OCIOSA_MINUTOS_T3	: DINT;
	num_MAQUINA_OCIOSA_HORAS_T3		: DINT;
	
	
	//CONTADORES
	time_SEGUNDOS					: INT;
	time_MINUTOS					: INT;
	time_HORAS						: INT;
	time_DIA						: INT;
	time_MES						: INT;
	time_ANO						: INT;
	
	bit_HORARIO_MINUTO_COMPLETO		: BOOL;
	bit_HORARIO_HORA_COMPLETO		: BOOL;
	bit_HORARIO_DIA_COMPLETO		: BOOL;
	bit_HORARIO_DIA_COMPLETO_REAL	: BOOL;
	bit_CONTADORES_RESET			: BOOL;
	
	num_PILHAS_COMPLETADAS_T1		: LREAL;
	num_PILHAS_COMPLETADAS_T2		: LREAL;
	num_PILHAS_COMPLETADAS_T3		: LREAL;
	
	num_PILHAS_REJEITADAS_T1		: LREAL;
	num_PILHAS_REJEITADAS_T2		: LREAL;
	num_PILHAS_REJEITADAS_T3		: LREAL;
	
	num_PILHAS_TOTAL_T1				: LREAL;
	num_PILHAS_TOTAL_T2				: LREAL;
	num_PILHAS_TOTAL_T3				: LREAL;

	
	tmr_MAQUINA_RODANDO_T1			: DINT;
	tmr_MAQUINA_RODANDO_T2			: DINT;
	tmr_MAQUINA_RODANDO_T3			: DINT;
	
	tmr_MAQUINA_PARADA_T1			: DINT;
	tmr_MAQUINA_PARADA_T2			: DINT;
	tmr_MAQUINA_PARADA_T3			: DINT;
	
	tmr_MAQUINA_OCIOSA_T1			: DINT;
	tmr_MAQUINA_OCIOSA_T2			: DINT;
	tmr_MAQUINA_OCIOSA_T3			: DINT;
	
	
	num_PORCENTAGEM_COMPLETADAS_T1 			: REAL;
	num_PORCENTAGEM_COMPLETADAS_T2 			: REAL;
	num_PORCENTAGEM_COMPLETADAS_T3 			: REAL;
	num_PORCENTAGEM_REJEITADAS_T1			: REAL;
	num_PORCENTAGEM_REJEITADAS_T2 			: REAL;
	num_PORCENTAGEM_REJEITADAS_T3 			: REAL;
	
	ihm_HIST_PORCENTAGEM_COMPLETADAS_T1		: DINT;
	ihm_HIST_PORCENTAGEM_COMPLETADAS_T2		: DINT;
	ihm_HIST_PORCENTAGEM_COMPLETADAS_T3		: DINT;
	ihm_HIST_PORCENTAGEM_REJEITADAS_T1		: DINT;
	ihm_HIST_PORCENTAGEM_REJEITADAS_T2		: DINT;
	ihm_HIST_PORCENTAGEM_REJEITADAS_T3		: DINT;
	
	
	info_DIA_ANTERIOR				: DINT;
	info_MES_ANTERIOR				: DINT;
	
	turno_A							: BOOL;
	turno_B							: BOOL;
	turno_C							: BOOL;
	
	ihm_HIST_INDEX_TURNO1			: ARRAY[0..9] OF BOOL;
	ihm_HIST_INDEX_TURNO2			: ARRAY[0..9] OF BOOL;
	ihm_HIST_INDEX_TURNO3			: ARRAY[0..9] OF BOOL;
	
	
	
	ONS_DIA_COMPLETO_1				: R_TRIG;;
	
	
//COP DIA 1
	COP_ihm_DIA_TURNO				: COP;
	COP_ihm_DIA_TURNO_AUX			: COP;
	
	COP_ihm_MES_TURNO				: COP;
	COP_ihm_MES_TURNO_AUX			: COP;
	
	COP_ihm_RODANDO_TURNO			: COP;
	COP_ihm_RODANDO_TURNO_AUX		: COP;
	
	COP_ihm_PARADO_TURNO			: COP;
	COP_ihm_PARADO_TURNO_AUX		: COP;
	
	COP_ihm_OCIOSO_TURNO			: COP;
	COP_ihm_OCIOSO_TURNO_AUX		: COP;

	COP_ihm_PILHAS_COMPLETADAS_TURNO		: COP;
	COP_ihm_PILHAS_COMPLETADAS_TURNO_AUX	: COP;	
	
	COP_ihm_PILHAS_REJEITADAS_TURNO			: COP;
	COP_ihm_PILHAS_REJEITADAS_TURNO_AUX		: COP;	
	
	COP_ihm_PILHAS_TOTAL_TURNO				: COP;
	COP_ihm_PILHAS_TOTAL_TURNO_AUX			: COP;	

	
	COP_ihm_PORCENTAGEM_COMPLETADAS			: COP;
	COP_ihm_PORCENTAGEM_COMPLETADAS_AUX		: COP;
	
	COP_ihm_PORCENTAGEM_REJEITADAS			: COP;
	COP_ihm_PORCENTAGEM_REJEITADAS_AUX		: COP;
	
	
//COP DIA 2
	COP_ihm_DIA_TURNO2				: COP;
	COP_ihm_DIA_TURNO_AUX2			: COP;
	
	COP_ihm_MES_TURNO2				: COP;
	COP_ihm_MES_TURNO_AUX2			: COP;
	
	COP_ihm_RODANDO_TURNO2			: COP;
	COP_ihm_RODANDO_TURNO_AUX2		: COP;
	
	COP_ihm_PARADO_TURNO2			: COP;
	COP_ihm_PARADO_TURNO_AUX2		: COP;
	
	COP_ihm_OCIOSO_TURNO2			: COP;
	COP_ihm_OCIOSO_TURNO_AUX2		: COP;

	COP_ihm_PILHAS_COMPLETADAS_TURNO2		: COP;
	COP_ihm_PILHAS_COMPLETADAS_TURNO_AUX2	: COP;	
	
	COP_ihm_PILHAS_REJEITADAS_TURNO2		: COP;
	COP_ihm_PILHAS_REJEITADAS_TURNO_AUX2	: COP;	
	
	COP_ihm_PILHAS_TOTAL_TURNO2				: COP;
	COP_ihm_PILHAS_TOTAL_TURNO_AUX2			: COP;	

	
	COP_ihm_PORCENTAGEM_COMPLETADAS2		: COP;
	COP_ihm_PORCENTAGEM_COMPLETADAS_AUX2	: COP;
	
	COP_ihm_PORCENTAGEM_REJEITADAS2			: COP;
	COP_ihm_PORCENTAGEM_REJEITADAS_AUX2		: COP;
	
	
//COP DIA 3
	COP_ihm_DIA_TURNO3				: COP;
	COP_ihm_DIA_TURNO_AUX3			: COP;
	
	COP_ihm_MES_TURNO3				: COP;
	COP_ihm_MES_TURNO_AUX3			: COP;
	
	COP_ihm_RODANDO_TURNO3			: COP;
	COP_ihm_RODANDO_TURNO_AUX3		: COP;
	
	COP_ihm_PARADO_TURNO3			: COP;
	COP_ihm_PARADO_TURNO_AUX3		: COP;
	
	COP_ihm_OCIOSO_TURNO3			: COP;
	COP_ihm_OCIOSO_TURNO_AUX3		: COP;

	COP_ihm_PILHAS_COMPLETADAS_TURNO3		: COP;
	COP_ihm_PILHAS_COMPLETADAS_TURNO_AUX3	: COP;	
	
	COP_ihm_PILHAS_REJEITADAS_TURNO3		: COP;
	COP_ihm_PILHAS_REJEITADAS_TURNO_AUX3	: COP;	
	
	COP_ihm_PILHAS_TOTAL_TURNO3				: COP;
	COP_ihm_PILHAS_TOTAL_TURNO_AUX3			: COP;	

	
	COP_ihm_PORCENTAGEM_COMPLETADAS3		: COP;
	COP_ihm_PORCENTAGEM_COMPLETADAS_AUX3	: COP;
	
	COP_ihm_PORCENTAGEM_REJEITADAS3			: COP;
	COP_ihm_PORCENTAGEM_REJEITADAS_AUX3		: COP;
	
	
	HORARIO_ATUAL_ANO				: YEAR;
	HORARIO_ATUAL_MES				: MONTH;
	HORARIO_ATUAL_DIA				: DAY;
	HORARIO_ATUAL_HORA				: HOUR;
	HORARIO_ATUAL_MINUTO			: MINUTE;
	HORARIO_ATUAL_SEGUNDO			: SECOND;
	
//BITS ATUADORES MODO MANUAL

	//ESTEIRAS DO EMPILHAMENTO DE SACOLA
	est_ROLETES_GIRO_MESA					: BOOL;
	est_INSPECAO_EMPILHADOR 				: BOOL;
	est_ROLETES_GIRO_MESA_REVERSE			: BOOL;
	est_INSPECAO_EMPILHADOR_REVERSE			: BOOL;

	//ESTEIRAS DO ENVOLVEDOR
	est_ENVOLVEDOR_ENTRADA					: BOOL;
	est_TRANSPORTADOR_ENVOLVEDOR			: BOOL;
	est_ENVOLVEDOR_SAIDA					: BOOL;
	
	//ESTEIRAS PARA REALIZAR PESAGEM DE SACOLAS
	est_MESA_DE_TRANSFERENCIA				: BOOL;
	est_REJEITO_PRODUTO						: BOOL;
	est_TRANSPORTADOR_PESAGEM				: BOOL;
	est_TRANSPORTADOR_ESTAGIO_1				: BOOL;
	est_TRANNSPORTADOR_MERGER				: BOOL;
	est_MESA_DE_TRANSFERENCIA_REVERSE		: BOOL;
	est_TRANSPORTADOR_PESAGEM_REVERSE		: BOOL;
	
	//BITS DE SELEÇÃO DE ATUADOR
	int_EMPILHADOR_ATUADOR_SELECIONADO		: INT;
	int_ENVOLVEDOR_ATUADOR_SELECIONADO		: INT;
	int_PESAGEM_ATUADOR_SELECIONADO			: INT;
	
	bit_ATU_EMPILHADOR_AVANCADO				: BOOL;
	bit_ATU_EMPILHADOR_RECUADO				: BOOL;
	bit_ATU_EMPILHADOR_AVANCAR				: BOOL;
	bit_ATU_EMPILHADOR_RECUAR				: BOOL;
	
	bit_ATU_ENVOLVEDOR_AVANCADO				: BOOL;
	bit_ATU_ENVOLVEDOR_RECUADO				: BOOL;
	bit_ATU_ENVOLVEDOR_AVANCAR				: BOOL;
	bit_ATU_ENVOLVEDOR_RECUAR				: BOOL;
	
	bit_ATU_PESAGEM_AVANCADO				: BOOL;
	bit_ATU_PESAGEM_RECUADO					: BOOL;
	bit_ATU_PESAGEM_AVANCAR					: BOOL;
	bit_ATU_PESAGEM_RECUAR					: BOOL;
	
	//SELECIONAR ATUADORES EMPILHADOR
	bit_SELEC_EMPILHADOR_GARRA_SACOLA		: BOOL;
	bit_SELEC_EMPILHADOR_BANDEJA			: BOOL;
	bit_SELEC_EMPILHADOR_DESCE_MESA_GIRO	: BOOL;
	bit_SELEC_EMPILHADOR_POSICIONA_SACOLA	: BOOL;
	
	//SELECIONAR ATUADORES ENVOLVEDOR
	bit_SELEC_ENVOLVEDOR_APROX_GARRA		: BOOL;
	bit_SELEC_ENVOLVEDOR_GARRA_DUPLA		: BOOL;
	bit_SELEC_ENVOLVEDOR_CORTE_FILME		: BOOL;
	bit_SELEC_ENVOLVEDOR_VACUO_FILME		: BOOL;
	bit_SELEC_ENVOLVEDOR_FECHA_FILME_1		: BOOL;
	bit_SELEC_ENVOLVEDOR_FECHA_FILME_2		: BOOL;
	bit_SELEC_ENVOLVEDOR_FECHA_FILME_3		: BOOL;
	
	
	//SELECIONAR ATUADORES PESAGEM
	bit_SELEC_PESAGEM_ACIONAMENTO_TRANSFERENCIA		: BOOL;

	
	bit_EMPILHA_SACOLA_HOME: BOOL;
	bit_bt_RESET_INSPECAO		: BOOL;
	bit_bt_RESET_EST_ENTRADA	: BOOL;
	bit_bt_RESET_EST_TR			: BOOL;
	bit_bt_RESET_EST_SAIDA		: BOOL;
	bit_ENV_CORTE_FILME		: BOOL;
	bit_bt_RESET_PESAGEM		: BOOL;
	
	
	bit_PORTA_1								: BOOL;
	bit_PORTA_2								: BOOL;
	bit_ATU_POSICIONADOR_AVANCADO: BOOL;
	bit_ATU_POSICIONADOR_RECUADO: BOOL;
	bit_ATU_POSICIONADOR_AVANCAR: BOOL;
	bit_ATU_POSICIONADOR_RECUAR: BOOL;
	
	
	//HISTÓRICO DE PESO
	hist_VALOR_PESAGEM_ARRAY				: ARRAY[0..9] OF REAL;
	hist_VALOR_PESAGEM_ARRAY_AUX			: ARRAY[0..9] OF REAL;
	cop_HIST_PESAGEM						: COP;
	cop_HIST_PESAGEM_AUX					: COP;
	
END_VAR

// TESTES_IOS
PROGRAM TESTES_IOS
VAR
END_VAR

// 	//E-16LA_EMP.diO - SLOT 1 (RMT50001)	
// 		LA_EMP.di_SENS_MESA_GIRO_RC				;
// 		LA_EMP.di_SENS_MESA_GIRO_MD				;
// 		LA_EMP.di_SENS_PINCA_GARRA_EMPILHADOR_RC	;
// 		LA_EMP.di_SENS_APOIO_BANDEJA_RC			;
// 		LA_EMP.di_SENS_EST_INSPEC_PRODUTO_1		;
// 		LA_EMP.di_SENS_MESA_GIRO_AV				;
// 		LA_EMP.di_SENS_PINCA_GARRA_EMPILHADOR_AV	;
// 		LA_EMP.di_SENS_APOIO_BANDEJA_AV			;
// 		LA_EMP.di_SENS_PRODUTO_MESA_GIRO			;
// 		LA_EMP.di_SENS_EST_INSPEC_PRODUTO_2		;




// 		LA_EMP.do_ATU_MESA_GIRO_RC				: BOOL;
// 		LA_EMP.do_ATU_PINCA_GARRA_EMPILHADOR	: BOOL;
// 		LA_EMP.do_ATU_MESA_GIRO_AV				: BOOL;
// 		LA_EMP.do_ATU_BANDEJA_APOIO			
// 		
// 	//E-16LA_EMP.diO - SLOT 2 (RMT50002)	
// 		LA_EMP.di_feedback_ERRO_MESA_GIRO			;
// 		LA_EMP.di_feedback_ERRO_EST_INSPECAO		;
//

END_PROGRAM

// DATA_TYPE/COP
FUNCTION_BLOCK COP

VAR_INPUT
  Source : POINTER TO DINT;  (* ADR(source[0]) convertido para POINTER TO BYTE *)
  Dest   : POINTER TO DINT;  (* ADR(dest[0]) convertido para POINTER TO BYTE *)
  Length    : UDINT;            (* nº de elementos a copiar *)
  Trigger   : BOOL;             (* sinal para fazer pulso *)
END_VAR

VAR
  prevTrig  : R_TRIG;    (* detecta borda de subida *)
  i         : UDINT;
END_VAR

(* Detect rising edge *)
IF prevTrig.Q  THEN
 

    (* Cópia elemento-a-elemento *)
    FOR i := 0 TO Length - 1 DO
      Dest[i] := Source[i];
      
    END_FOR;

    
  END_IF;


(* armazena estado do trigger para próxima varredura *)
prevTrig(CLK:= Trigger);

END_FUNCTION_BLOCK

// DATA_TYPE/FB_ATUADOR
FUNCTION_BLOCK FB_ATUADOR

VAR_INPUT
	in_SAFETY_ATIVO		: BOOL;
	in_MODO_MANUAL		: BOOL;
	in_AUTO_CMD			: BOOL;
	in_MANUAL_CMD		: BOOL;
	in_SENSORIAMENTO	: INT; // Tipo de Sensoriamento (0: Sem sensores; 1: Apenas RC; 2: Apenas AV; 3: RC e AV)
	in_SENSOR_RC		: BOOL;
	in_SENSOR_AV		: BOOL;
END_VAR

VAR_OUTPUT
	out_VALVULA_RC		: BOOL;
	out_VALVULA_AV		: BOOL;
	out_ALARME_AV		: BOOL;
	out_ALARME_RC		: BOOL;
END_VAR

VAR
	bit_CMD_ATUADOR		: BOOL;
	tmr_ALARME_AV		: TON;
	tmr_ALARME_RC		: TON;
END_VAR

//	COMANDO		============//============//============//============//============//============//============
// Seleciona a fonte do comando conforme o modo

	IF in_SAFETY_ATIVO THEN

		IF in_MODO_MANUAL THEN
			bit_CMD_ATUADOR := in_MANUAL_CMD;
		ELSE
			bit_CMD_ATUADOR := in_AUTO_CMD;
		END_IF
	
		out_VALVULA_AV := bit_CMD_ATUADOR;
		out_VALVULA_RC := NOT bit_CMD_ATUADOR;
		
	END_IF
	
//	ALARMES		============//============//============//============//============//============//============
// 	Alarme dispara se a válvula estiver comandada e o sensor correspondente não confirmar a posição dentro do tempo.

CASE in_SENSORIAMENTO	OF
		
0:	// Sem sensores
	out_ALARME_AV	:= FALSE;
	out_ALARME_RC	:= FALSE;
	
1: 	//Apenas Sensor Recuado
	tmr_ALARME_RC (PT	:= T#2000MS, IN	:= in_SAFETY_ATIVO	AND out_VALVULA_RC AND NOT in_SENSOR_RC);
	out_ALARME_RC	:= tmr_ALARME_RC.Q;
	
	out_ALARME_AV	:= FALSE;
	
2:	//Apenas Sensor Avançado
	out_ALARME_RC	:= FALSE;
	
	tmr_ALARME_AV (PT	:= T#2000MS, IN	:= in_SAFETY_ATIVO	AND out_VALVULA_AV AND NOT in_SENSOR_AV);
	out_ALARME_AV	:= tmr_ALARME_AV.Q;
	
3:	// Sensor Recuado e Avançado
	tmr_ALARME_RC (PT	:= T#2000MS, IN	:= in_SAFETY_ATIVO	AND out_VALVULA_RC AND NOT in_SENSOR_RC);
	out_ALARME_RC	:= tmr_ALARME_RC.Q;
	
	tmr_ALARME_AV (PT	:= T#2000MS, IN	:= in_SAFETY_ATIVO	AND out_VALVULA_AV AND NOT in_SENSOR_AV);
	out_ALARME_AV	:= tmr_ALARME_AV.Q;	
	
END_CASE

END_FUNCTION_BLOCK

// LADO_A/01 - LA_GERAL/ALARMES
PROGRAM ALARMES
VAR
	tmr_alarm_1000		:	TON;
	tmr_alarm_1001		:	TON;
	tmr_alarm_1002		:	TON;
	tmr_alarm_1003		:	TON;
	tmr_alarm_1004		:	TON;
	tmr_alarm_1005		:	TON;
	tmr_alarm_1006		:	TON;
	tmr_alarm_1007		:	TON;
	tmr_alarm_1008		:	TON;
	tmr_alarm_1009		:	TON;
	tmr_alarm_1010		:	TON;
	tmr_alarm_1011		:	TON;
	tmr_alarm_1012		:	TON;
	tmr_alarm_1013		:	TON;
	tmr_alarm_1014		:	TON;
	tmr_alarm_1015		:	TON;
	tmr_alarm_1016		:	TON;
	tmr_alarm_1017		:	TON;
	tmr_alarm_1018		:	TON;
	tmr_alarm_1019		:	TON;
	tmr_alarm_1020		:	TON;
	tmr_alarm_1021		:	TON;
	tmr_alarm_1022		:	TON;
	tmr_alarm_1023		:	TON;
	tmr_alarm_1024		:	TON;
	tmr_alarm_1025		:	TON;
	tmr_alarm_1026		:	TON;
	tmr_alarm_1027		:	TON;
	tmr_alarm_1028		:	TON;
	
END_VAR

// //ATIVAÇÃO DE ÍCONE DE ALARME
// IF 		GVL_CELULA.status_alarm_EIXO_Y 	 		 > 0	OR
// 		GVL_CELULA.status_alarm_EIXO_Z 	 		 > 0 	OR
// 		GVL_CELULA.status_alarm_EIXO_COLMEIA_1	 > 0	OR 
// 		GVL_CELULA.status_alarm_EIXO_COLMEIA_2	 > 0	OR
// 		GVL_CELULA.status_alarm_HOME_EIXO_Y		 > 0	OR
// 		GVL_CELULA.status_alarm_HOME_EIXO_Z		 > 0	OR
// 		GVL_CELULA.status_alarm_HOME_DIVERTER		 > 0	OR
// 		GVL_CELULA.status_alarm_atu_DIVERTER_FREIO > 0 	OR 
// 		GVL_CELULA.status_alarm_atu_FORM_EMPURADDOR > 0	OR
// 		GVL_CELULA.status_alarm_atu_FORM_FORMADOR	 > 0	OR
// 		GVL_CELULA.status_alarm_atu_FORM_PEGA_CAIXA > 0 	OR
// 		GVL_CELULA.status_alarm_atu_FORM_VACUO	 > 0	OR
// 		GVL_CELULA.status_alarm_atu_MANI_GARRA	 > 0	OR
// 		GVL_CELULA.status_alarm_atu_POSICIONA_PRODUTO > 0 OR
// 		GVL_CELULA.status_alarm_atu_PRODUTO_FREIO	 > 0 	OR
// 		GVL_CELULA.status_alarm_atu_SEPARADOR_Y	 > 0 	OR
// 		GVL_CELULA.status_alarm_atu_SEPARADOR_Z	 > 0 	OR
// 		GVL_CELULA.status_alarm_atu_STOP_ENTREGA	 > 0 	OR
// 		GVL_CELULA.status_alarm_atu_STOP_PRE_ENTREGA > 0	OR
// 		GVL_CELULA.status_alarm_SAFETY_CASE		 > 0	OR
// 		GVL_CELULA.status_alarm_SAFETY_FORM		 > 0	OR
// 		GVL_CELULA.status_alarm_in_PORTA_CASE_1	 > 0	OR
// 		GVL_CELULA.status_alarm_in_PORTA_CASE_2	 > 0	OR
// 		GVL_CELULA.status_alarm_in_PORTA_CASE_3	 > 0	OR
// 		GVL_CELULA.status_alarm_in_PORTA_CASE_4	 > 0	OR
// 		GVL_CELULA.status_alarm_in_PORTA_CASE_5	 > 0	OR
// 		GVL_CELULA.status_alarm_in_PORTA_DIVERTER  > 0	OR
// 		GVL_CELULA.status_alarm_ACUMULO_CAIXAS	 > 0	OR
// 		GVL_CELULA.status_alarm_FALTA_CAIXA		 > 0	OR
// 		GVL_CELULA.status_alarm_TEMP_COLA			 > 0	OR
// 		GVL_CELULA.status_alarm_NIVEL_COLA		 > 0	OR
// 		GVL_CELULA.status_alarm_VACUO_COLMEIA		 > 0	OR
// 		GVL_CELULA.status_alarm_BRACO_COLMEIA		 > 0	OR
// 		GVL_CELULA.status_alarm_INDEX_CAIXAS		 > 0	OR
// 		GVL_CELULA.status_alarm_COLMEIA_FREIO		 > 0	THEN
// 			
// 			GVL_IHM.ALARME_ATIVO	:=	TRUE;
// 	ELSE
// 			GVL_IHM.ALARME_ATIVO	:=	FALSE;
// 	END_IF
// 	
// 	
// 		IF bt_MAQUINA_RESET THEN
// 		GVL_CELULA.status_alarm_EIXO_Y 	 		 := 0; 
// 		GVL_CELULA.status_alarm_EIXO_Z 	 		 := 0; 
// 		GVL_CELULA.status_alarm_EIXO_COLMEIA_1	 := 0; 
// 		GVL_CELULA.status_alarm_EIXO_COLMEIA_2	 := 0; 
// 		GVL_CELULA.status_alarm_HOME_EIXO_Y		 := 0;
// 		GVL_CELULA.status_alarm_HOME_EIXO_Z		 := 0;
// 		GVL_CELULA.status_alarm_HOME_DIVERTER		 := 0;
// 		GVL_CELULA.status_alarm_atu_DIVERTER_FREIO := 0; 
// 		GVL_CELULA.status_alarm_atu_FORM_EMPURADDOR := 0;
// 		GVL_CELULA.status_alarm_atu_FORM_FORMADOR	 := 0;
// 		GVL_CELULA.status_alarm_atu_FORM_PEGA_CAIXA := 0;
// 		GVL_CELULA.status_alarm_atu_FORM_VACUO	 := 0;
// 		GVL_CELULA.status_alarm_atu_MANI_GARRA	 := 0;
// 		GVL_CELULA.status_alarm_atu_POSICIONA_PRODUTO := 0;
// 		GVL_CELULA.status_alarm_atu_PRODUTO_FREIO	 := 0;
// 		GVL_CELULA.status_alarm_atu_SEPARADOR_Y	 := 0;
// 		GVL_CELULA.status_alarm_atu_SEPARADOR_Z	 := 0;
// 		GVL_CELULA.status_alarm_atu_STOP_ENTREGA	 := 0;
// 		GVL_CELULA.status_alarm_atu_STOP_PRE_ENTREGA := 0;
// 		GVL_CELULA.status_alarm_SAFETY_CASE		 := 0;
// 		GVL_CELULA.status_alarm_SAFETY_FORM		 := 0;
// 		GVL_CELULA.status_alarm_in_PORTA_CASE_1	 := 0;
// 		GVL_CELULA.status_alarm_in_PORTA_CASE_2	 := 0;
// 		GVL_CELULA.status_alarm_in_PORTA_CASE_3	 := 0;
// 		GVL_CELULA.status_alarm_in_PORTA_CASE_4	 := 0;
// 		GVL_CELULA.status_alarm_in_PORTA_CASE_5	 := 0;
// 		GVL_CELULA.status_alarm_in_PORTA_DIVERTER  := 0;
// 		GVL_CELULA.status_alarm_ACUMULO_CAIXAS	 := 0;
// 		GVL_CELULA.status_alarm_FALTA_CAIXA		 := 0;
// 		GVL_CELULA.status_alarm_NIVEL_COLA		 := 0;
// 		GVL_CELULA.status_alarm_TEMP_COLA			 := 0;
// 		GVL_CELULA.status_alarm_VACUO_COLMEIA		 := 0;
// 		GVL_CELULA.status_alarm_BRACO_COLMEIA		 := 0;
// 		GVL_CELULA.status_alarm_INDEX_CAIXAS		 := 0;
// 		GVL_CELULA.status_alarm_COLMEIA_FREIO		 := 0;
// 	END_IF
// 	
// 	
// 	
// 
// 
// 
// 
// //ALARMES DE ATUADORES DURANTE O PROCESSO	
// IF GVL_CELULA.bit_SAFETY_ATIVO THEN
// 	
// //EXPANSÃO DO STOP ENTREGA
// 		tmr_alarm_1000 (IN	:= atu_STOP_ENTREGA_RC	AND NOT	sens_ATU_STOP_ENTREGA_RC, PT := T#2S);
// 		tmr_alarm_1001 (IN	:= atu_STOP_ENTREGA_AV	AND NOT	sens_ATU_STOP_ENTREGA_AV, PT := T#2S);
// 		
// 		IF	tmr_alarm_1000.Q			THEN
// 					GVL_CELULA.status_alarm_atu_STOP_ENTREGA	:= 1;
// 		ELSIF tmr_alarm_1001.Q			THEN
// 					GVL_CELULA.status_alarm_atu_STOP_ENTREGA	:= 2;
// 		ELSE
// 					GVL_CELULA.status_alarm_atu_STOP_ENTREGA	:= 0;
// 		END_IF
// 		
// 		
// //EXPANSÃO DO STOP PRE ENTREGA
// 	//	tmr_alarm_1002 (IN	:= atu_STOP_PRE_ENTREGA_RC	AND NOT	sens_ATU_STOP_PRE_ENTREGA_AV, PT := T#2S);
// 		tmr_alarm_1003 (IN	:= atu_STOP_PRE_ENTREGA_AV	AND NOT	sens_ATU_STOP_PRE_ENTREGA_RC, PT := T#2S);
// 		
// 		IF	tmr_alarm_1002.Q			THEN
// 					GVL_CELULA.status_alarm_atu_STOP_PRE_ENTREGA	:= 1;
// 		ELSIF tmr_alarm_1003.Q			THEN
// 					GVL_CELULA.status_alarm_atu_STOP_PRE_ENTREGA	:= 2;
// 		ELSE
// 					GVL_CELULA.status_alarm_atu_STOP_PRE_ENTREGA	:= 0;
// 		END_IF
// 			
// 
// //EXPANSÃO DO FREIO DE PRODUTOS
// 		tmr_alarm_1006 (IN	:= atu_PRODUTO_FREIO_RC	AND NOT	sens_ATU_PRODUTO_FREIO_RC, PT := T#2S);
// 		tmr_alarm_1007 (IN	:= atu_PRODUTO_FREIO_AV	AND NOT	sens_ATU_PRODUTO_FREIO_AV, PT := T#2S);
// 		
// 		IF	tmr_alarm_1006.Q			THEN
// 					GVL_CELULA.status_alarm_atu_PRODUTO_FREIO	:= 1;
// 		ELSIF tmr_alarm_1007.Q			THEN
// 					GVL_CELULA.status_alarm_atu_PRODUTO_FREIO	:= 2;
// 		ELSE
// 					GVL_CELULA.status_alarm_atu_PRODUTO_FREIO	:= 0;
// 		END_IF
// 
// 		
// //EXPANSÃO DO SEPARADOR Y
// 		tmr_alarm_1008 (IN	:= atu_SEPARADOR_Y_RC	AND NOT	sens_ATU_SEPARADOR_Y_RC, PT := T#2S);
// 		tmr_alarm_1009 (IN	:= atu_SEPARADOR_Y_AV	AND NOT	sens_ATU_SEPARADOR_Y_AV, PT := T#2S);
// 		
// 	(*	IF	tmr_alarm_1008.Q			THEN
// 					GVL_CASE.status_alarm_atu_SEPARADOR_Y	:= 1;
// 		ELSIF tmr_alarm_1009.Q			THEN
// 					GVL_CASE.status_alarm_atu_SEPARADOR_Y	:= 2;
// 		ELSE
// 					GVL_CASE.status_alarm_atu_SEPARADOR_Y	:= 0;
// 		END_IF*)
// 		
// 		
// //EXPANSÃO DO SEPARADOR Z
// 		tmr_alarm_1010 (IN	:= atu_SEPARADOR_Z_RC	AND NOT	sens_ATU_SEPARADOR_Z_RC, PT := T#2S);
// 		tmr_alarm_1011 (IN	:= atu_SEPARADOR_Z_AV	AND NOT	sens_ATU_SEPARADOR_Z_AV, PT := T#2S);
// 		
// 		IF	tmr_alarm_1010.Q			THEN
// 					GVL_CELULA.status_alarm_atu_SEPARADOR_Z	:= 1;
// 		ELSIF tmr_alarm_1011.Q			THEN
// 					GVL_CELULA.status_alarm_atu_SEPARADOR_Z	:= 2;
// 		ELSE
// 					GVL_CELULA.status_alarm_atu_SEPARADOR_Z	:= 0;
// 		END_IF
// 		
// 		
// //EXPANSÃO DO FREIO DO DIVERTER
// 		tmr_alarm_1012 (IN	:= atu_DIVERTER_FREIO_RC	AND NOT	sens_ATU_DIVERTER_FREIO_RC, PT := T#2S);
// 		tmr_alarm_1013 (IN	:= atu_DIVERTER_FREIO_AV	AND NOT	sens_ATU_DIVERTER_FREIO_AV, PT := T#2S);
// 		
// 		IF	tmr_alarm_1012.Q			THEN
// 					GVL_CELULA.status_alarm_atu_DIVERTER_FREIO	:= 1;
// 		ELSIF tmr_alarm_1013.Q			THEN
// 					GVL_CELULA.status_alarm_atu_DIVERTER_FREIO	:= 2;
// 		ELSE
// 					GVL_CELULA.status_alarm_atu_DIVERTER_FREIO	:= 0;
// 		END_IF
// 		
// 	
// //EXPANSÃO DO PEGADOR
// 		tmr_alarm_1014 (IN	:= valv_FORM_PEGA_CAIXA_RC	AND NOT sens_FORM_PEGADOR_RC, PT := T#2S);
// 		tmr_alarm_1015 (IN	:= valv_FORM_PEGA_CAIXA_AV	AND NOT	sens_FORM_PEGADOR_AV, PT := T#2S);
// 		
// 		IF	tmr_alarm_1014.Q			THEN
// 					GVL_CELULA.status_alarm_atu_FORM_PEGA_CAIXA	:= 1;
// 		ELSIF tmr_alarm_1015.Q			THEN
// 					GVL_CELULA.status_alarm_atu_FORM_PEGA_CAIXA	:= 2;
// 		ELSE
// 					GVL_CELULA.status_alarm_atu_FORM_PEGA_CAIXA	:= 0;
// 		END_IF
// 		
// 		
// //EXPANSÃO DO FORMADOR
// 		tmr_alarm_1016 (IN	:= valv_FORM_FORMADOR_CAIXA_RC	AND NOT sens_ATU_FORMADOR_RC, PT := T#2S);
// 		tmr_alarm_1017 (IN	:= valv_FORM_FORMADOR_CAIXA_AV	AND NOT	sens_ATU_FORMADOR_AV, PT := T#2S);
// 		
// 		IF	tmr_alarm_1016.Q			THEN
// 					GVL_CELULA.status_alarm_atu_FORM_FORMADOR	:= 1;
// 		ELSIF tmr_alarm_1017.Q			THEN
// 					GVL_CELULA.status_alarm_atu_FORM_FORMADOR	:= 2;
// 		ELSE
// 					GVL_CELULA.status_alarm_atu_FORM_FORMADOR	:= 0;
// 		END_IF
// 			
// 		
// //EXPANSÃO DO EMPURRADOR
// 		tmr_alarm_1018 (IN	:= NOT valv_FORM_EMPURADDOR	AND NOT sens_ATU_EMPURRADOR_RC, PT := T#2S);
// 		tmr_alarm_1019 (IN	:= valv_FORM_EMPURADDOR		AND NOT	sens_ATU_EMPURRADOR_AV, PT := T#2S);
// 		
// 		IF	tmr_alarm_1018.Q			THEN
// 					GVL_CELULA.status_alarm_atu_FORM_EMPURADDOR	:= 1;
// 		ELSIF tmr_alarm_1019.Q			THEN
// 					GVL_CELULA.status_alarm_atu_FORM_EMPURADDOR	:= 2;
// 		ELSE
// 					GVL_CELULA.status_alarm_atu_FORM_EMPURADDOR	:= 0;
// 		END_IF
// 		
// 		
// //EXPANSÃO DO BRAÇO COLMEIA
// 		tmr_alarm_1023 (IN	:= atu_GARRA_COLMEIA_RC	AND NOT	sens_ATU_COLMEIA_BRACO_RC, PT := T#2S);
// 		tmr_alarm_1024 (IN	:= atu_GARRA_COLMEIA_AV	AND NOT	sens_ATU_COLMEIA_BRACO_AV, PT := T#2S);
// 		
// 		IF	tmr_alarm_1023.Q			THEN
// 					GVL_CELULA.status_alarm_BRACO_COLMEIA	:= 1;
// 		ELSIF tmr_alarm_1024.Q			THEN
// 					GVL_CELULA.status_alarm_BRACO_COLMEIA	:= 2;
// 		ELSE
// 					GVL_CELULA.status_alarm_BRACO_COLMEIA	:= 0;
// 		END_IF
// 		
// 	
// //EXPANSÃO DO INDEX CAIXAS
// 		tmr_alarm_1025 (IN	:= atu_CASE_INDEX_CAIXAS_RC	AND NOT	sens_ATU_COLMEIA_INDEX_RC, PT := T#2S);
// 		tmr_alarm_1026 (IN	:= atu_CASE_INDEX_CAIXAS_AV	AND NOT sens_ATU_COLMEIA_INDEX_AV, PT := T#2S);
// 		
// 		IF	tmr_alarm_1025.Q			THEN
// 					GVL_CELULA.status_alarm_INDEX_CAIXAS	:= 1;
// 		ELSIF tmr_alarm_1026.Q			THEN
// 					GVL_CELULA.status_alarm_INDEX_CAIXAS	:= 2;
// 		ELSE
// 					GVL_CELULA.status_alarm_INDEX_CAIXAS	:= 0;
// 		END_IF
// 		
// 		
// //EXPANSÃO DO INDEX CAIXAS
// 		tmr_alarm_1025 (IN	:= NOT 	atu_CASE_COLMEIA_FREIO_AV	AND NOT	sens_ATU_COLMEIA_FREIO_RC, PT := T#2S);
// 		tmr_alarm_1026 (IN	:= 		atu_CASE_COLMEIA_FREIO_AV	AND NOT sens_ATU_COLMEIA_FREIO_AV, PT := T#2S);
// 		
// 		IF	tmr_alarm_1025.Q			THEN
// 					GVL_CELULA.status_alarm_COLMEIA_FREIO	:= 1;
// 		ELSIF tmr_alarm_1026.Q			THEN
// 					GVL_CELULA.status_alarm_COLMEIA_FREIO	:= 2;
// 		ELSE
// 					GVL_CELULA.status_alarm_COLMEIA_FREIO	:= 0;
// 		END_IF
// 		
// //VACUO PRODUTO
// 		IF	GVL_MANI.BIT_ALARME_PEGA_PRODUTO		THEN
// 					GVL_CELULA.status_alarm_VACUO_PRODUTOS	:= 1;
// 		ELSE
// 					GVL_CELULA.status_alarm_VACUO_PRODUTOS	:= 0;
// 		END_IF
// 		
// //VACUO COLMEIA
// 		IF	GVL_COLMEIA.bit_ALARME_PEGA_COLMEIA		THEN
// 					GVL_CELULA.status_alarm_VACUO_COLMEIA	:= 1;
// 		ELSE
// 					GVL_CELULA.status_alarm_VACUO_COLMEIA	:= 0;
// 		END_IF
// 
// 		
// //FALTA DE CAIXAS NO SENSOR DE ACUMULO DE ENTRADA
// 		IF	GVL_CELULA.bit_ALARME_FALTA_CAIXA_ATIVO		THEN
// 					GVL_CELULA.status_alarm_FALTA_CAIXA	:= 1;
// 		ELSE
// 					GVL_CELULA.status_alarm_FALTA_CAIXA	:= 0;
// 		END_IF
// 		
// 		
// 		
// //ATIVAÇÃO DO VÁCUO
// 		tmr_alarm_1020 (IN	:= valv_FORM_VACUO	AND NOT sens_FORM_VACUOSTATO, PT := T#2S);
// 		
// 		IF	tmr_alarm_1020.Q			THEN
// 					GVL_CELULA.status_alarm_atu_FORM_FORMADOR	:= 1;
// 		ELSE
// 					GVL_CELULA.status_alarm_atu_FORM_FORMADOR	:= 0;
// 		END_IF
// 
// END_IF
// 
// 
// 
// //ALARME EIXO Y
// 		IF (GVL_IHM_CP.bit_EIXO_Y_ALARME_ATIVO OR NOT M00_EIXO_Y.bit_HABILITADO) AND GVL_CELULA.bit_SAFETY_ATIVO	THEN
// 			GVL_CELULA.status_alarm_EIXO_Y	:= 1;
// 		ELSE	
// 			GVL_CELULA.status_alarm_EIXO_Y	:= 0;
// 		END_IF
// 		
// //ALARME EIXO Z
// 		IF (GVL_IHM_CP.bit_EIXO_Z_ALARME_ATIVO OR NOT M01_EIXO_Z.bit_HABILITADO) AND GVL_CELULA.bit_SAFETY_ATIVO THEN
// 			GVL_CELULA.status_alarm_EIXO_Z	:= 1;
// 		ELSE	
// 			GVL_CELULA.status_alarm_EIXO_Z	:= 0;
// 		END_IF
// 		
// //ALARME DIVERTER
// 		IF (GVL_IHM_CP.bit_DIVERTER_ALARME_ATIVO OR NOT M02_DIVERTER.bit_HABILITADO) AND GVL_CELULA.bit_SAFETY_ATIVO	THEN
// 			GVL_CELULA.status_alarm_DIVERTER	:= 1;
// 		ELSE	
// 			GVL_CELULA.status_alarm_DIVERTER	:= 0;
// 		END_IF
// 		
// //ALARME EIXO COLMEIA 1
// 		IF (GVL_IHM_CP.bit_EIXO_COLMEIA_1_ALARME_ATIVO) AND GVL_CELULA.bit_SAFETY_ATIVO	THEN
// 			GVL_CELULA.status_alarm_EIXO_COLMEIA_1	:= 1;
// 		ELSE	
// 			GVL_CELULA.status_alarm_EIXO_COLMEIA_1	:= 0;
// 		END_IF
// 		
// //ALARME EIXO COLMEIA 2
// 		IF (GVL_IHM_CP.bit_EIXO_COLMEIA_2_ALARME_ATIVO) AND GVL_CELULA.bit_SAFETY_ATIVO	THEN
// 			GVL_CELULA.status_alarm_EIXO_COLMEIA_2	:= 1;
// 		ELSE	
// 			GVL_CELULA.status_alarm_EIXO_COLMEIA_2	:= 0;
// 		END_IF
// 		
// 	//ALARME HOME EIXO Y
// 		IF M00_EIXO_Y.bit_HOME_ERRO THEN
// 			GVL_CELULA.status_alarm_HOME_EIXO_Y	:=	1;
// 		ELSE
// 			GVL_CELULA.status_alarm_HOME_EIXO_Y	:=	0;
// 		END_IF
// 		
// //ALARME HOME EIXO Z
// 		IF M01_EIXO_Z.bit_HOME_ERRO THEN
// 			GVL_CELULA.status_alarm_HOME_EIXO_Z	:=	1;
// 		ELSE
// 			GVL_CELULA.status_alarm_HOME_EIXO_Z	:=	0;
// 		END_IF
// 		
// //ALARME HOME DIVERTER
// 		IF M02_DIVERTER.bit_HOME_ERRO THEN
// 			GVL_CELULA.status_alarm_HOME_DIVERTER	:=	1;
// 		ELSE
// 			GVL_CELULA.status_alarm_HOME_DIVERTER	:=	0;
// 		END_IF
// 		
// 		
// //ALARME EMERGÊNCIA CASE
// 		IF NOT in_SAFETY_ATIVO THEN
// 			GVL_CELULA.status_alarm_SAFETY_CASE	:=	1;
// 		ELSE
// 			GVL_CELULA.status_alarm_SAFETY_CASE	:=	0;
// 		END_IF
// 		
// 		
// //ALARME EMERGÊNCIA CASE
// 		IF NOT in_SAFETY_ATIVO_FORM THEN
// 			GVL_CELULA.status_alarm_SAFETY_FORM	:=	1;
// 		ELSE
// 			GVL_CELULA.status_alarm_SAFETY_FORM	:=	0;
// 		END_IF
// 		
// //ALARME PALETIZADOR NÃO RODANDO
// 		(*IF NOT PALETIZADOR_OUT.bit_PALETIZADOR_MAQUINA_RODANDO AND NOT
// 			PALETIZADOR_OUT.bit_FORCE_CASEPACKER THEN
// 			GVL_CASE.status_alarm_PL_RODANDO	:=	1;
// 		ELSE
// 			GVL_CASE.status_alarm_PL_RODANDO	:=	0;
// 		END_IF*)
// 		
// 		
// //ALARME ACUMULO PRODUTOS
// 		IF GVL_PRODUTOS.bit_ACUMULO_PRODUTOS_ALARME	THEN
// 			GVL_CELULA.status_alarm_ACUMULO_COPOS	 := 1;
// 		ELSE
// 			GVL_CELULA.status_alarm_ACUMULO_COPOS	 := 0;
// 		END_IF
// 		
// //ALARME ACUMULO CAIXAS
// 		IF GVL_CAIXAS.bit_CAIXA_SAIDA_ACUMULO	THEN
// 			GVL_CELULA.status_alarm_ACUMULO_CAIXAS  := 1;
// 		ELSE
// 			GVL_CELULA.status_alarm_ACUMULO_CAIXAS  := 0;
// 		END_IF	
// 		
// //FALTA NO PEGADOR DE CAIXAS DA FORMADORA
// 		IF	GVL_FORM.bit_FALHA_PEGADOR		THEN
// 					GVL_CELULA.status_alarm_FALHA_PEGA	:= 1;
// 		ELSE
// 					GVL_CELULA.status_alarm_FALHA_PEGA	:= 0;
// 		END_IF
// 		
// //FALTA DE COLMEIAS
// 		IF	GVL_COLMEIA.bit_FALTANDO_CAIXAS		THEN
// 					GVL_CELULA.status_alarm_NIVEL_COLMEIA	:= 1;
// 		ELSE
// 					GVL_CELULA.status_alarm_NIVEL_COLMEIA	:= 0;
// 		END_IF
// 		
// 		
// //ALARME SEM PRESSÃO NA LINHA E COM SAFETY ATIVO
// 		IF in_FEEDBACK_AR_1 AND GVL_CELULA.bit_SAFETY_ATIVO THEN
// 			tmr_alarm_1022.IN						:= TRUE;
// 		ELSE
// 			tmr_alarm_1022.IN						:= FALSE;
// 		END_IF
// 		
// 		IF tmr_alarm_1022.Q THEN
// 			GVL_CELULA.status_alarm_AR			 	:= 1;
// 			GVL_CELULA.bit_ALARME_AR_CASE_ATIVO	:= TRUE;
// 		ELSE
// 			GVL_CELULA.status_alarm_AR			 	:= 0;
// 			GVL_CELULA.bit_ALARME_AR_CASE_ATIVO	:= FALSE;
// 		END_IF
// 		
// tmr_alarm_1022(PT:= T#3S);
// 		
// //ALARME TEMPERATURA COLEIRO
// 		IF NOT in_COLA_TEMP_OK AND NOT in_NIVEL_COLA_FALHA THEN
// 			GVL_CELULA.status_alarm_TEMP_COLA  := 1;
// 			GVL_FORM.bit_FALHA_COLA_TEMP	 := 1;
// 		ELSE
// 			GVL_CELULA.status_alarm_TEMP_COLA  := 0;
// 			GVL_FORM.bit_FALHA_COLA_TEMP	 := 0;
// 		END_IF
// 		
// //ALARME NIVEL DE COLA COLEIRO
// 		IF  in_NIVEL_COLA_FALHA	THEN
// 			GVL_CELULA.status_alarm_NIVEL_COLA  := 1;
// 			GVL_FORM.bit_FALHA_COLA_NIVEL	  := 1;
// 		ELSE
// 			GVL_CELULA.status_alarm_NIVEL_COLA  := 0;
// 			GVL_FORM.bit_FALHA_COLA_NIVEL	  := 0;
// 		END_IF
// 
// 
// //ALARME PORTAS
// 		IF  NOT GVL_IHM_CP.bit_CASE_PORTA_1 THEN
// 			GVL_CELULA.status_alarm_in_PORTA_CASE_1	:=	1;
// 		ELSE
// 			GVL_CELULA.status_alarm_in_PORTA_CASE_1	:=	0;
// 		END_IF
// 		
// 		IF  NOT GVL_IHM_CP.bit_CASE_PORTA_2 THEN
// 			GVL_CELULA.status_alarm_in_PORTA_CASE_2	:=	1;
// 		ELSE
// 			GVL_CELULA.status_alarm_in_PORTA_CASE_2	:=	0;
// 		END_IF
// 		
// 		IF  NOT GVL_IHM_CP.bit_CASE_PORTA_3 THEN
// 			GVL_CELULA.status_alarm_in_PORTA_CASE_3	:=	1;
// 		ELSE
// 			GVL_CELULA.status_alarm_in_PORTA_CASE_3	:=	0;
// 		END_IF
// 		
// 		IF  NOT GVL_IHM_CP.bit_CASE_PORTA_4 THEN
// 			GVL_CELULA.status_alarm_in_PORTA_CASE_4	:=	1;
// 		ELSE
// 			GVL_CELULA.status_alarm_in_PORTA_CASE_4	:=	0;
// 		END_IF
// 		
// 		IF  NOT GVL_IHM_CP.bit_CASE_PORTA_5 THEN
// 			GVL_CELULA.status_alarm_in_PORTA_CASE_5	:=	1;
// 		ELSE
// 			GVL_CELULA.status_alarm_in_PORTA_CASE_5	:=	0;
// 		END_IF
// 		
// 	//	IF  NOT GVL_IHM_CP.bit_CASE_PORTA_DIVERTER THEN
// 	//		GVL_CASE.status_alarm_in_PORTA_DIVERTER	:=	1;
// 	//	ELSE
// 	//		GVL_CASE.status_alarm_in_PORTA_DIVERTER	:=	0;
// 	//	END_IF
// 		
// 		IF  NOT GVL_IHM_CP.bit_FORM_PORTA_1 THEN
// 			GVL_CELULA.status_alarm_in_PORTA_FORM_1	:=	1;
// 		ELSE
// 			GVL_CELULA.status_alarm_in_PORTA_FORM_1	:=	0;
// 		END_IF
// 		
// 		IF  NOT GVL_IHM_CP.bit_FORM_PORTA_2 THEN
// 			GVL_CELULA.status_alarm_in_PORTA_FORM_2	:=	1;
// 		ELSE
// 			GVL_CELULA.status_alarm_in_PORTA_FORM_2	:=	0;
// 		END_IF
// 		
// 		IF  NOT GVL_IHM_CP.bit_FORM_PORTA_3 THEN
// 			GVL_CELULA.status_alarm_in_PORTA_FORM_3	:=	1;
// 		ELSE
// 			GVL_CELULA.status_alarm_in_PORTA_FORM_3	:=	0;
// 		END_IF
// 		
// 		
// 		
// //ALARME BOTÕES DE EMERGÊNCIA
// 
// 		IF NOT bt_EMERGENCIA_CASE_1	THEN
// 			GVL_CELULA.status_alarm_BT_EMERGENCIA_CASE_1	:=	1;
// 		ELSE
// 			GVL_CELULA.status_alarm_BT_EMERGENCIA_CASE_1	:=	0;
// 		END_IF
// 		
// 		IF NOT bt_EMERGENCIA_CASE_2	THEN
// 			GVL_CELULA.status_alarm_BT_EMERGENCIA_CASE_2	:=	1;
// 		ELSE
// 			GVL_CELULA.status_alarm_BT_EMERGENCIA_CASE_2	:=	0;
// 		END_IF
// 		
// 		IF NOT bt_EMERGENCIA_FORM	THEN
// 			GVL_CELULA.status_alarm_BT_EMERGENCIA_FORM	:=	1;
// 		ELSE
// 			GVL_CELULA.status_alarm_BT_EMERGENCIA_FORM	:=	0;
// 		END_IF
//

END_PROGRAM

// DATA_TYPE/FB_Markem_SelecionarMacro
FUNCTION_BLOCK FB_Markem_SelecionarMacro
VAR_INPUT
    // Habilita a conexão TCP
    xEnable : BOOL;

    // Pulso para selecionar uma macro
    xSelecionar : BOOL;

    // Nome da macro, sem extensão
    sNomeMacro : STRING(24);
END_VAR

VAR_OUTPUT
    // Conexão estabelecida com a Markem
    xConnected : BOOL;

    // Envio em andamento
    xBusy : BOOL;

    // Pulso de conclusão
    xDone : BOOL;

    // Erro geral
    xError : BOOL;

    // Última macro enviada
    sUltimaMacroEnviada : STRING(24);

    // Diagnósticos da biblioteca
    eErroCliente : NBS.ERROR;
    eErroEscrita : NBS.ERROR;
END_VAR

VAR
    // Comunicação CAA
    fbTCPClient : NBS.TCP_Client;
    fbTCPWrite  : NBS.TCP_Write;

    // Endereço IP da impressora
    stIPMarkem : NBS.IP_ADDR :=
        (sAddr := '192.168.0.40');

    // Handle entregue pelo TCP_Client
    hConnectionMarkem : CAA.HANDLE :=
        CAA.gc_hINVALID;

    // Controle interno
    xClienteAtivo : BOOL;
    xExecuteWrite : BOOL;
    xErroInterno  : BOOL;

    // Telegrama
    sBufferTX : STRING(100);
    szTamanhoTX : CAA.SIZE;

    // Nome memorizado durante o envio
    sMacroPendente : STRING(24);

    // Máquina de estados
    uiEstado : UINT;

    // Borda de subida
    rtSelecionar : R_TRIG;
END_VAR

// Pulso de apenas um ciclo
xDone := FALSE;

// Borda de subida para selecionar a macro
rtSelecionar(CLK := xSelecionar);


// ============================================================
// CLIENTE TCP
// ============================================================

// Entrada herdada do CBM.LTrig
fbTCPClient.xEnable := xEnable;

fbTCPClient(
    udiTimeOut  := UDINT#5_000_000,
    ipAddr      := stIPMarkem,
    uiPort      := UINT#9100,
    eError      => eErroCliente,
    xActive     => xClienteAtivo,
    hConnection => hConnectionMarkem
);

xConnected := xClienteAtivo;


// ============================================================
// MÁQUINA DE ESTADOS
// ============================================================

IF NOT xEnable THEN

    uiEstado := 0;
    xExecuteWrite := FALSE;
    xBusy := FALSE;
    xErroInterno := FALSE;

ELSE

    CASE uiEstado OF

        // ----------------------------------------------------
        // Estado 0: aguardando comando
        // ----------------------------------------------------
        0:
            xExecuteWrite := FALSE;
            xBusy := FALSE;

            IF rtSelecionar.Q THEN

                xErroInterno := FALSE;

                IF xClienteAtivo
                   AND (LEN(sNomeMacro) > 0) THEN

                    // Memoriza o nome para que não mude
                    // durante o envio
                    sMacroPendente := sNomeMacro;

                    // Monta:
                    // !M "40x50"<CR>
                    sBufferTX := CONCAT(
                        '!M "',
                        sMacroPendente
                    );

                    sBufferTX := CONCAT(
                        sBufferTX,
                        '"$R'
                    );

                    // Converte o tamanho para CAA.SIZE
                    szTamanhoTX :=
                        CAA.UDINT_TO_SIZE(
                            TO_UDINT(LEN(sBufferTX))
                        );

                    // Gera borda de subida no TCP_Write
                    xExecuteWrite := TRUE;
                    xBusy := TRUE;

                    uiEstado := 10;

                ELSE

                    xErroInterno := TRUE;

                END_IF;

            END_IF;


        // ----------------------------------------------------
        // Estado 10: aguardando o envio terminar
        // ----------------------------------------------------
        10:
            xExecuteWrite := TRUE;
            xBusy := TRUE;

            IF fbTCPWrite.xDone THEN

                xExecuteWrite := FALSE;
                xBusy := FALSE;

                sUltimaMacroEnviada :=
                    sMacroPendente;

                xDone := TRUE;

                uiEstado := 20;

            ELSIF fbTCPWrite.xError THEN

                xExecuteWrite := FALSE;
                xBusy := FALSE;
                xErroInterno := TRUE;

                uiEstado := 20;

            ELSIF NOT xClienteAtivo THEN

                xExecuteWrite := FALSE;
                xBusy := FALSE;
                xErroInterno := TRUE;

                uiEstado := 20;

            END_IF;


        // ----------------------------------------------------
        // Estado 20: reseta o TCP_Write
        // ----------------------------------------------------
        20:
            // O TCP_Write precisa receber FALSE depois
            // da conclusão para poder detectar uma nova borda
            xExecuteWrite := FALSE;
            xBusy := FALSE;

            uiEstado := 0;


        ELSE

            uiEstado := 0;
            xExecuteWrite := FALSE;
            xBusy := FALSE;

    END_CASE;

END_IF;


// ============================================================
// ESCRITA TCP
// ============================================================

// Entradas herdadas do CBM.ETrigTo
fbTCPWrite.xExecute := xExecuteWrite;
fbTCPWrite.udiTimeOut := UDINT#0;

fbTCPWrite(
    hConnection := hConnectionMarkem,
    szSize       := szTamanhoTX,
    pData        := ADR(sBufferTX),
    eError       => eErroEscrita
);


// ============================================================
// DIAGNÓSTICO GERAL
// ============================================================

xError :=
    xErroInterno
    OR fbTCPClient.xError
    OR fbTCPWrite.xError;

END_FUNCTION_BLOCK

// DATA_TYPE/FB_SMARTMOTOR
FUNCTION_BLOCK FB_SMARTMOTOR

VAR_INPUT
	in_SAFETY_ATIVO			: BOOL;
	in_MODO_MANUAL			: BOOL;
	in_AUTO_CMD_FWD			: BOOL;
	in_AUTO_CMD_REV			: BOOL;
	in_MANUAL_CMD_FWD		: BOOL;
	in_MANUAL_CMD_REV		: BOOL;
	in_FALHA_MOTOR			: BOOL;
	in_RESET_ALARME			: BOOL;
END_VAR

VAR_OUTPUT
	out_MOTOR_FWD			: BOOL;
	out_MOTOR_REV			: BOOL;
	out_ALARME				: BOOL;
END_VAR

VAR
	bit_CMD_FWD				: BOOL;
	bit_CMD_REV				: BOOL;
	sr_FALHA				: SR;
END_VAR

//	COMANDO		============//============//============//============//============//============//============
	// Seleciona a fonte do comando conforme o modo
	// Motor desliga se safety inativa OU alarme de falha travado
	
	IF in_SAFETY_ATIVO AND NOT in_FALHA_MOTOR THEN

		IF in_MODO_MANUAL THEN
			bit_CMD_FWD := in_MANUAL_CMD_FWD;
			bit_CMD_REV := in_MANUAL_CMD_REV;
		ELSE
			bit_CMD_FWD := in_AUTO_CMD_FWD;
			bit_CMD_REV := in_AUTO_CMD_REV;
		END_IF

		// Intertravamento: nunca aciona FWD e REV simultaneamente
		out_MOTOR_FWD := bit_CMD_FWD AND NOT bit_CMD_REV;
		out_MOTOR_REV := bit_CMD_REV AND NOT bit_CMD_FWD;

	ELSE
		// Safety inativa ou falha do motor: desliga o motor
		out_MOTOR_FWD := FALSE;
		out_MOTOR_REV := FALSE;

	END_IF

//	FALHA		============//============//============//============//============//============//============
	// Falha só é considerada válida com a segurança ativa.
	// Uma vez travada, só sai com in_RESET_ALARME (reset manual do operador).

	sr_FALHA (SET1 := in_SAFETY_ATIVO AND in_FALHA_MOTOR, RESET := in_RESET_ALARME);
	out_ALARME	 := sr_FALHA.Q1;

END_FUNCTION_BLOCK

// DATA_TYPE/LEITURA_DATA_PLC
PROGRAM LEITURA_DATA_PLC
VAR
	UTC_time_in_ms: SYSTIME;
	loc_time_str: SYSTIMEDATE;
	loc_time_in_ms: SYSTIME;
	local_date_time: DATE_AND_TIME;
	Local_TOD: TIME_OF_DAY;
	time_teste: DATE_AND_TIME;
	bool_teste: BOOL;
	SetDateAndTime_Teste: RTCLK.SetDateAndTime;
	teste: BOOL;
	RTON_0: RTON;
	MUDAR_DATA: DATE_AND_TIME;
END_VAR

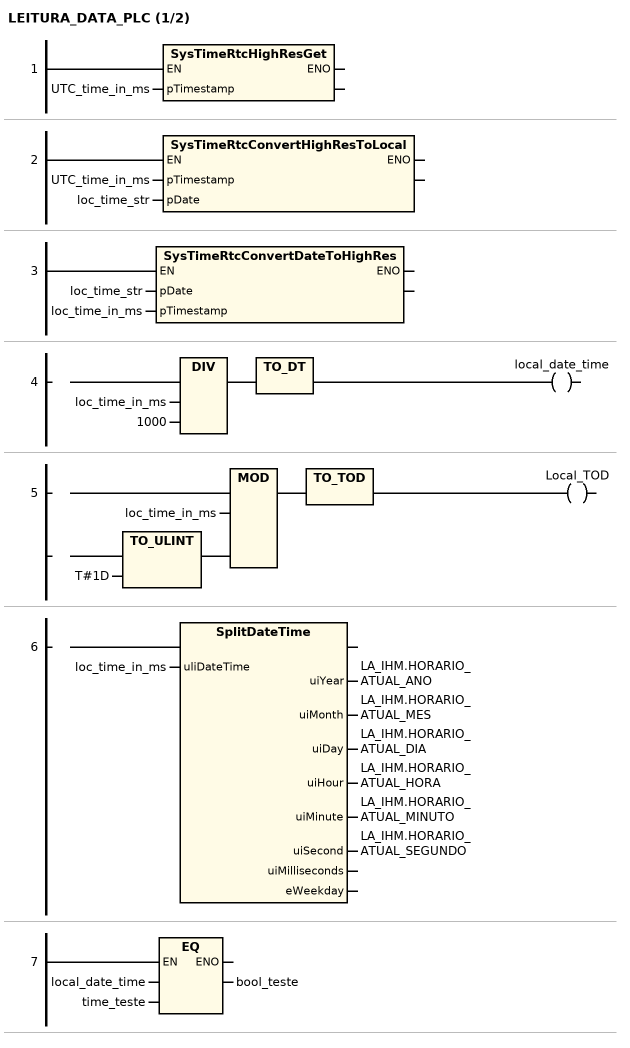
// NETWORK 1
SysTimeRtcHighResGet(pTimestamp := UTC_time_in_ms);

// NETWORK 2
SysTimeRtcConvertHighResToLocal(pTimestamp := UTC_time_in_ms, pDate := loc_time_str);

// NETWORK 3
SysTimeRtcConvertDateToHighRes(pDate := loc_time_str, pTimestamp := loc_time_in_ms);

// NETWORK 4
local_date_time := TO_DT(loc_time_in_ms / 1000);

// NETWORK 5
Local_TOD := TO_TOD(loc_time_in_ms MOD TO_ULINT(T#1D));

// NETWORK 6
SplitDateTime(uliDateTime := loc_time_in_ms, uiYear => LA_IHM.HORARIO_ATUAL_ANO, uiMonth => LA_IHM.HORARIO_ATUAL_MES, uiDay => LA_IHM.HORARIO_ATUAL_DIA, uiHour => LA_IHM.HORARIO_ATUAL_HORA, uiMinute => LA_IHM.HORARIO_ATUAL_MINUTO, uiSecond => LA_IHM.HORARIO_ATUAL_SEGUNDO);

// NETWORK 7
bool_teste := local_date_time = time_teste;

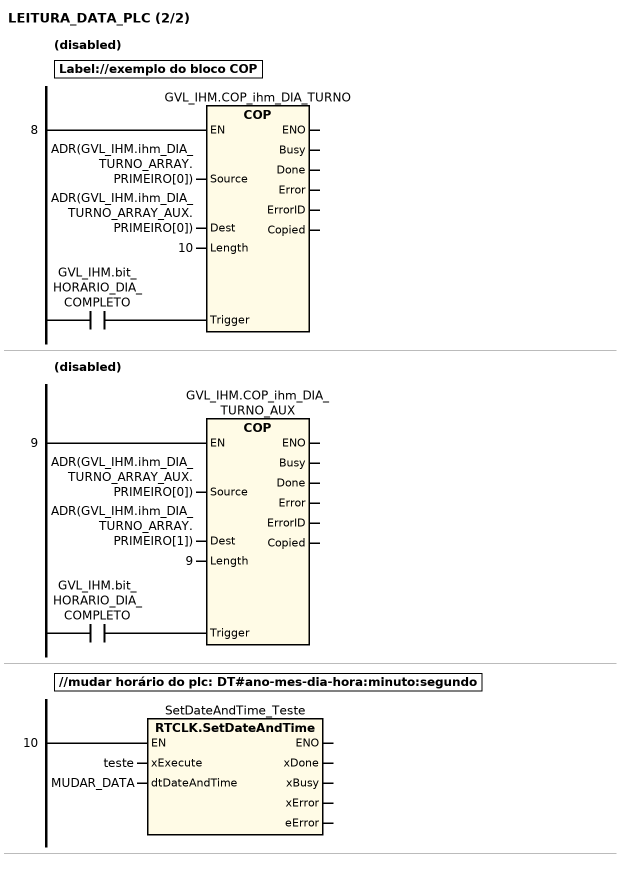
// NETWORK 8 (disabled)
// label: Label://exemplo do bloco COP
// GVL_IHM.COP_ihm_DIA_TURNO(
//     Source := ADR(GVL_IHM.ihm_DIA_TURNO_ARRAY.PRIMEIRO[0]),
//     Dest := ADR(GVL_IHM.ihm_DIA_TURNO_ARRAY_AUX.PRIMEIRO[0]),
//     Length := 10,
//     Trigger := GVL_IHM.bit_HORARIO_DIA_COMPLETO); // COP

// NETWORK 9 (disabled)
// GVL_IHM.COP_ihm_DIA_TURNO_AUX(
//     Source := ADR(GVL_IHM.ihm_DIA_TURNO_ARRAY_AUX.PRIMEIRO[0]),
//     Dest := ADR(GVL_IHM.ihm_DIA_TURNO_ARRAY.PRIMEIRO[1]),
//     Length := 9,
//     Trigger := GVL_IHM.bit_HORARIO_DIA_COMPLETO); // COP

// NETWORK 10
// label: //mudar horário do plc: DT#ano-mes-dia-hora:minuto:segundo
SetDateAndTime_Teste(xExecute := teste, dtDateAndTime := MUDAR_DATA); // RTCLK.SetDateAndTime

END_PROGRAM

// DATA_TYPE/RTON
FUNCTION_BLOCK RTON
VAR_INPUT
	T_IN		: BOOL	:=	FALSE;
	T_PT		: TIME;
	Timer_reset	: BOOL;	
END_VAR
VAR_OUTPUT
	RTON_Out	: BOOL;
	RTON_ET		: TIME;
END_VAR
VAR
	TON_0		: TON;
	T_ET		: TIME;
	F_TRIG_0	: F_TRIG;
	R_TRIG_0	: R_TRIG;
	T_PT_Tmp	: TIME;
	RTON_ET_Tmp	: TIME;
END_VAR
VAR // added by the converter: edge detectors and wires of the graphical bodies
    _w1, _w2 : BOOL;
END_VAR

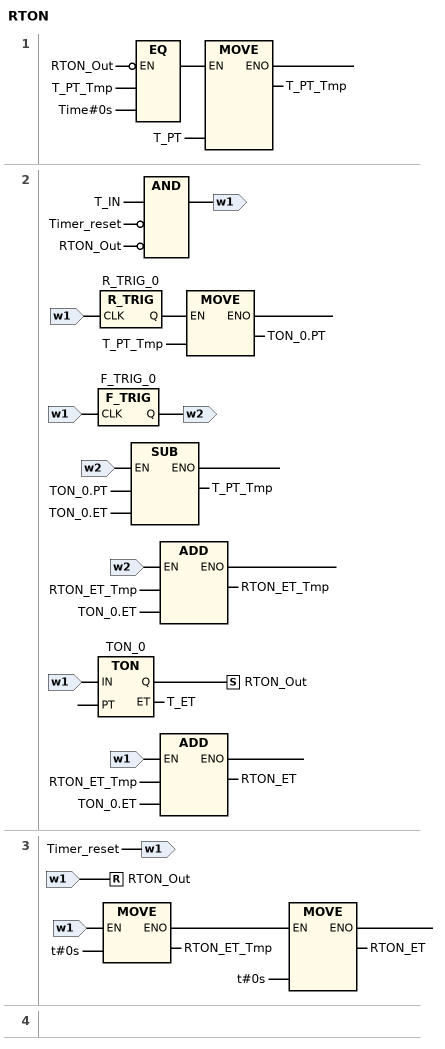
// NETWORK 1
IF NOT RTON_Out AND T_PT_Tmp = Time#0s THEN T_PT_Tmp := T_PT; END_IF

// NETWORK 2
_w1 := T_IN AND NOT Timer_reset AND NOT RTON_Out;
R_TRIG_0(CLK := _w1); // R_TRIG
IF R_TRIG_0.Q THEN TON_0.PT := T_PT_Tmp; END_IF
F_TRIG_0(CLK := _w1); // F_TRIG
IF F_TRIG_0.Q THEN T_PT_Tmp := TON_0.PT - TON_0.ET; END_IF
IF F_TRIG_0.Q THEN RTON_ET_Tmp := RTON_ET_Tmp + TON_0.ET; END_IF
TON_0(IN := _w1, ET => T_ET); // TON
RTON_Out S= TON_0.Q;
IF _w1 THEN RTON_ET := RTON_ET_Tmp + TON_0.ET; END_IF

// NETWORK 3
RTON_Out R= Timer_reset;
_w2 := Timer_reset;
IF _w2 THEN RTON_ET_Tmp := t#0s; END_IF
IF _w2 THEN RTON_ET := t#0s; END_IF

// NETWORK 4

END_FUNCTION_BLOCK

// D_PESAGEM/D00_PESAGEM
PROGRAM D00_PESAGEM
VAR
	reset_rotina		: BOOL;
	bit_SHIFT_HIST_PESO : BOOL;
	passo_PESAGEM		: INT := 9;
	
	f_trig_ENTRADA	:	F_TRIG;
	f_trig_SAIDA	:	F_TRIG;
	
	tmr_TRANSFERINDO_PILHA			: TON;
	tmr_PARADA_ESTEIRA				: TON;
	tmr_VERIFICA_PESO				: TON;
	TESTE: BOOL;
END_VAR


IF LA_IHM.bit_bt_RESET_PESAGEM	THEN
	passo_PESAGEM	:=	9;
END_IF



CASE passo_PESAGEM OF
	
//--------------------------------------------------------------------------------------------------------------------------------------------------------------------------------
09://reset rotina

	GVL_PESAGEM.bit_valv_ACIONAMENTO_TRANSFERENCIA	:=	TRUE;
	GVL_PESAGEM.est_TRANSPORTADOR_PESAGEM			:=	FALSE;
	GVL_PESAGEM.est_TRANSPORTADOR_PESAGEM_REVERSE	:=	FALSE;
	GVL_PESAGEM.est_REJEITO_PRODUTO					:=	FALSE;
	GVL_PESAGEM.est_MESA_DE_TRANSFERENCIA_REVERSE	:=	FALSE;
	GVL_PESAGEM.est_MESA_DE_TRANSFERENCIA			:=	FALSE;
	bit_SHIFT_HIST_PESO								:= 	FALSE;
	LA_IHM.bit_STATUS_PESAGEM						:=	0;
	
	est_BALANCA										:=	FALSE;
	est_BALANCA_REVERSE								:=	FALSE;
	
	passo_PESAGEM	:=	10;
	
	
//--------------------------------------------------------------------------------------------------------------------------------------------------------------------------------
10://aguarda feedback de sensor de avanço

	IF sens_TRANSFERENCIA_AV THEN
		GVL_PESAGEM.bit_PESANDO_PILHA_SACOLA := FALSE;
		passo_PESAGEM						 :=	999;
	END_IF


//--------------------------------------------------------------------------------------------------------------------------------------------------------------------------------
999://inicia ciclo com máquina rodando e sem processo de pesagem de sacola iniciado

	IF (LA_GERAL.bit_MAQUINA_RODANDO OR TESTE) AND NOT GVL_PESAGEM.bit_PESANDO_PILHA_SACOLA	THEN
		passo_PESAGEM				:=	1000;
		LA_IHM.bit_STATUS_PESAGEM	:=	0;
	END_IF
	
	
//--------------------------------------------------------------------------------------------------------------------------------------------------------------------------------
1000://decide em qual direção ligar a esteira de transferencia baseado na prioridade de recebimento de lado da esteira de saída do envolvedor

	IF LA_ENV.bit_ENVOLVEDOR_ENVIANDO_PILHA THEN
		GVL_PESAGEM.est_MESA_DE_TRANSFERENCIA_REVERSE	:=	FALSE;
		GVL_PESAGEM.bit_ENVOLVEDOR_1					:=	TRUE;
		GVL_PESAGEM.bit_ENVOLVEDOR_2					:=	FALSE;
		GVL_PESAGEM.est_MESA_DE_TRANSFERENCIA			:=	TRUE;
		passo_PESAGEM									:=	1001;
	ELSIF GVL_PESAGEM.bit_ENVOLVEDOR_ENVIANDO_PILHA_2 AND NOT LA_ENV.bit_ENVOLVEDOR_ENVIANDO_PILHA	THEN
		GVL_PESAGEM.est_MESA_DE_TRANSFERENCIA_REVERSE	:=	true;
		GVL_PESAGEM.bit_ENVOLVEDOR_1					:=	FALSE;
		GVL_PESAGEM.bit_ENVOLVEDOR_2					:=	TRUE;
		GVL_PESAGEM.est_MESA_DE_TRANSFERENCIA			:=	TRUE;
		passo_PESAGEM									:=	1001;
	END_IF
	
//--------------------------------------------------------------------------------------------------------------------------------------------------------------------------------
1001://declara inicio de processo de psagem da pilha de sacola para intertravamento de recebimento de pilha do lado 1 ou lado 2
	
	GVL_PESAGEM.bit_PESANDO_PILHA_SACOLA	:=	TRUE;
	passo_PESAGEM							:=	1002;
	
//--------------------------------------------------------------------------------------------------------------------------------------------------------------------------------
1002://aguarda tempo após acionar sensor para desligar esteira de transferência

	IF sens_MESA_TRANSFER_1 OR sens_MESA_TRANSFER_2	THEN
		tmr_TRANSFERINDO_PILHA.IN	:=	TRUE;
	END_IF
	
	IF tmr_TRANSFERINDO_PILHA.Q	THEN
		tmr_TRANSFERINDO_PILHA.IN						:=	FALSE;
		GVL_PESAGEM.est_MESA_DE_TRANSFERENCIA_REVERSE	:=	FALSE;
		GVL_PESAGEM.est_MESA_DE_TRANSFERENCIA			:=	FALSE;
		passo_PESAGEM									:=	1003;
	END_IF
	
	
//--------------------------------------------------------------------------------------------------------------------------------------------------------------------------------
1003://recua atuador de transferencia e aguarda feedback de sensor recuado

	GVL_PESAGEM.bit_valv_ACIONAMENTO_TRANSFERENCIA	:=	FALSE;

	IF sens_TRANSFERENCIA_RC	THEN
		passo_PESAGEM	:=	1004;
	END_IF
	
//--------------------------------------------------------------------------------------------------------------------------------------------------------------------------------
1004://Liga esteiraS de transferencia e da balança para transportar pilha para balança

	GVL_PESAGEM.est_TRANSPORTADOR_PESAGEM	:=	TRUE;
	est_BALANCA								:=	TRUE;
	est_BALANCA_REVERSE						:=	FALSE;
	LA_IHM.bit_STATUS_PESAGEM				:=	1;
	
	passo_PESAGEM							:=	1005;
	
//--------------------------------------------------------------------------------------------------------------------------------------------------------------------------------
1005: //espera confirmação de borda de descida de sensor de entrada da balança

	IF f_trig_ENTRADA.Q	THEN
		tmr_PARADA_ESTEIRA.IN		:= TRUE;
	END_IF
	
	IF	tmr_PARADA_ESTEIRA.Q	THEN
			tmr_PARADA_ESTEIRA.IN		:= FALSE;
			tmr_VERIFICA_PESO.IN		:= TRUE;
			est_BALANCA					:=	FALSE;
			passo_PESAGEM				:=	3000;
	END_IF
		
//--------------------------------------------------------------------------------------------------------------------------------------------------------------------------------
3000://verifica se peso atual está condizente com a receita 

	IF tmr_VERIFICA_PESO.Q	THEN
			GVL_PESAGEM.status_VALOR_PESAGEM		:= Peso_medido;
			LA_IHM.hist_VALOR_PESAGEM_ARRAY[0]	:=	Peso_medido;
			tmr_VERIFICA_PESO.IN					:= FALSE;
			passo_PESAGEM							:=	1006;
	END_IF
	
//--------------------------------------------------------------------------------------------------------------------------------------------------------------------------------
1006://verifica se peso atual está condizente com a receita 

	IF GVL_PESAGEM.bit_PESAGEM_OK THEN
		GVL_PESAGEM.bit_PESAGEM_ATUAL	:=	TRUE;
		GVL_PESAGEM.array_HIST_PESO.0	:=	FALSE;
		LA_IHM.bit_STATUS_PESAGEM		:=	2;
		passo_PESAGEM					:=	1007;
	ELSE
		GVL_PESAGEM.bit_PESAGEM_ERRO	:=	TRUE;
		GVL_PESAGEM.array_HIST_PESO.0	:=	TRUE;
		LA_IHM.bit_STATUS_PESAGEM		:=	3;
		passo_PESAGEM					:=	1008;
	END_IF
	
//--------------------------------------------------------------------------------------------------------------------------------------------------------------------------------
1007://caso peso esteja ok, aguarda borda de descida do sensor de saída da balança
	est_BALANCA					:=	TRUE;
	
	IF f_trig_SAIDA.Q	THEN
		passo_PESAGEM					:=	1009;
	END_IF
	
//--------------------------------------------------------------------------------------------------------------------------------------------------------------------------------
1008://caso peso esteja com erro, gira esteira da balança ao contrário

	est_BALANCA_REVERSE						:=	TRUE;
	passo_PESAGEM							:=	1009;

//--------------------------------------------------------------------------------------------------------------------------------------------------------------------------------
1009://Verifica feedback da balança. Se está OK, para a esteira e prepara para reinicio de ciclo. Se não, liga a esteira invertida e prepara para rejeito

	IF GVL_PESAGEM.bit_PESAGEM_ATUAL	THEN
		GVL_PESAGEM.est_TRANSPORTADOR_PESAGEM	:=	FALSE;
		est_BALANCA								:=	FALSE;
		GVL_PESAGEM.bit_PESAGEM_ATUAL				:=	FALSE;
		passo_PESAGEM							:=	1011;
	ELSIF GVL_PESAGEM.bit_PESAGEM_ERRO	THEN
		GVL_PESAGEM.est_TRANSPORTADOR_PESAGEM			:=	TRUE;
		GVL_PESAGEM.bit_ENVOLVEDOR_1					:=	FALSE;
		GVL_PESAGEM.bit_ENVOLVEDOR_2					:=	FALSE;
		GVL_PESAGEM.bit_PESAGEM_ERRO					:=	FALSE;
		GVL_PESAGEM.est_TRANSPORTADOR_PESAGEM_REVERSE	:=	TRUE;
		GVL_PESAGEM.est_REJEITO_PRODUTO					:=	TRUE;
		passo_PESAGEM									:=	1010;
	END_IF

//--------------------------------------------------------------------------------------------------------------------------------------------------------------------------------
1010://aguarda pilha chegar no final da esteira de rejeito para desligar esteiras

	IF sens_PRODUTO_REJEITO	THEN
		GVL_PESAGEM.est_TRANSPORTADOR_PESAGEM			:=	FALSE;
		GVL_PESAGEM.est_TRANSPORTADOR_PESAGEM_REVERSE	:=	FALSE;
		GVL_PESAGEM.est_REJEITO_PRODUTO					:=	FALSE;
		est_BALANCA_REVERSE								:=	FALSE;
		passo_PESAGEM									:=	1011;
	END_IF
	
	
//--------------------------------------------------------------------------------------------------------------------------------------------------------------------------------
1011://Desloca informações de peso e etiqueta

	GVL_PESAGEM.array_ETIQUETA		:=	SHL(GVL_PESAGEM.array_ETIQUETA, 1);
	GVL_PESAGEM.array_HIST_PESO		:=	SHL(GVL_PESAGEM.array_HIST_PESO, 1);
	bit_SHIFT_HIST_PESO				:=	TRUE;
	GVL_PESAGEM.array_HIST_PESO.0	:= 	FALSE;
	LA_IHM.bit_STATUS_PESAGEM		:=	0;
	passo_PESAGEM					:=	1012;
	
	
//--------------------------------------------------------------------------------------------------------------------------------------------------------------------------------
1012://aciona atuador de transferencia  e aguarda feedback do sensor de avanço para reiniciar ciclo e declarar que não está mais pesando sacola

	bit_SHIFT_HIST_PESO								:= FALSE;
	GVL_PESAGEM.bit_valv_ACIONAMENTO_TRANSFERENCIA	:= TRUE;
	
	IF sens_TRANSFERENCIA_AV	THEN
		GVL_PESAGEM.bit_PESANDO_PILHA_SACOLA := FALSE;
		LA_IHM.hist_VALOR_PESAGEM_ARRAY[0]	 := 0;
		passo_PESAGEM						 :=	999;
	END_IF

END_CASE





//------------//-----------LÓGICAS EXTRAS---------------//----------------------//--------------------------//

//-----------CHECAGEM DE PESO-------//--------------------//---------------------//

IF	Peso_medido	>= PVAR.rec_ATUAL.num_PESO_SACOLA - 500	AND
	Peso_medido	<= PVAR.rec_ATUAL.num_PESO_SACOLA + 500	THEN
			GVL_PESAGEM.bit_PESAGEM_OK	:= TRUE;
	ELSE
			GVL_PESAGEM.bit_PESAGEM_OK	:= FALSE;
	END_IF


//-----------ATUADORES-------------//--------------------//---------------------//

//ATUADOR TRANSFERENCIA PARA SEÇÃO DE PESAGEM
IF GVL_PESAGEM.bit_valv_ACIONAMENTO_TRANSFERENCIA	THEN
	valv_TRANSFERENCIA_RC	:=	FALSE;
	valv_TRANSFERENCIA_AV	:=	TRUE;
ELSE
	valv_TRANSFERENCIA_RC	:=	TRUE;
	valv_TRANSFERENCIA_AV	:=	FALSE;
END_IF


//DEFINE SE BIT DA PRIMEIRA CASA SERÁ TRUE OU FALSE PARA DECIDIR ETIQUETA
IF GVL_PESAGEM.bit_ENVOLVEDOR_1	THEN
		GVL_PESAGEM.array_ETIQUETA.0 :=	1;
ELSIF GVL_PESAGEM.bit_ENVOLVEDOR_2	THEN
		GVL_PESAGEM.array_ETIQUETA.0 :=	0;
END_IF


//HISTÓRICO DE VALOR DE PESO MEDIDO
LA_IHM.cop_HIST_PESAGEM(Source:= ADR(LA_IHM.hist_VALOR_PESAGEM_ARRAY[0]) , Dest:= ADR(LA_IHM.hist_VALOR_PESAGEM_ARRAY_AUX[0]), Length:= 10, Trigger:= bit_SHIFT_HIST_PESO);
LA_IHM.cop_HIST_PESAGEM_AUX(Source:= ADR(LA_IHM.hist_VALOR_PESAGEM_ARRAY_AUX[0]) , Dest:= ADR(LA_IHM.hist_VALOR_PESAGEM_ARRAY[1]), Length:= 9, Trigger:= bit_SHIFT_HIST_PESO);


//-----------TIMERS-------------//--------------------//---------------------//

tmr_TRANSFERINDO_PILHA(PT:= T#2.6S );
tmr_PARADA_ESTEIRA	(PT:= T#300MS);
tmr_VERIFICA_PESO	(PT:= T#1000MS);
f_trig_ENTRADA(CLK:= sens_ENTRADA_BALANCA);
f_trig_SAIDA(CLK:= sens_SAIDA_BALANCA);

END_PROGRAM

// D_PESAGEM/D01_EST_ETIQUETA
PROGRAM D01_EST_ETIQUETA
VAR
	reset_rotina	:	BOOL;
	passo_ETIQUETA	:	INT := 9;
	
	bit_ETIQUETA_PRONTA		:	BOOL;
	bit_ETIQUETA_IMPRIMINDO	:	BOOL;
	bit_ETIQUETA_CONCLUIDO	: 	BOOL;
	
	bit_IMPRIMIR_ETIQUETA_1	:	BOOL;
	bit_IMPRIMIR_ETIQUETA_2	:	BOOL;
	
	tmr_PARAR_ESTEIRA		:	TON;
	tmr_ETIQUETA			:	TON;
	TESTE: BOOL;
END_VAR


CASE passo_ETIQUETA OF
	
//--------------------------------------------------------------------------------------------------------------------------------------------------------------------------------
09://reset rotina

	bit_IMPRIMIR_ETIQUETA_1	:=	FALSE;
	bit_IMPRIMIR_ETIQUETA_2	:=	FALSE;
	tmr_ETIQUETA.IN			:=	FALSE;
	tmr_PARAR_ESTEIRA.IN	:=	FALSE;
	LA_GERAL.do_SAIDA_COLAR_EQUIQUETA	:=	FALSE;
	
	passo_ETIQUETA			:=	999;
	
	
//--------------------------------------------------------------------------------------------------------------------------------------------------------------------------------
999://inicia se a máquina estiver rodando

	IF LA_GERAL.bit_MAQUINA_RODANDO OR TESTE	THEN
		passo_ETIQUETA			:=	1000;
	END_IF

//--------------------------------------------------------------------------------------------------------------------------------------------------------------------------------
1000://Caso o feedback da balança corresponda como peso OK, liga esteira estagio 1

	IF GVL_PESAGEM.bit_PESAGEM_ATUAL	THEN
		GVL_PESAGEM.est_TRANSPORTADOR_ESTAGIO_1	:=	TRUE;
		passo_ETIQUETA			:=	1001;
	END_IF
	
//--------------------------------------------------------------------------------------------------------------------------------------------------------------------------------
1001://assim que chegar ao limite da esteira estágio 1, desliga a esteira

	IF sens_PRODUTO_BALANCA	THEN
		tmr_PARAR_ESTEIRA.IN	:=	TRUE;
	END_IF
	
	IF tmr_PARAR_ESTEIRA.Q	THEN
		tmr_PARAR_ESTEIRA.IN					:=	FALSE;
		GVL_PESAGEM.est_TRANSPORTADOR_ESTAGIO_1	:=	FALSE;
		LA_GERAL.do_SAIDA_COLAR_EQUIQUETA		:=	TRUE;
		passo_ETIQUETA							:=	1002;
	END_IF
	

//--------------------------------------------------------------------------------------------------------------------------------------------------------------------------------
1002://aguarda confirmação de que etiquetadora está operante
(*	IF bit_ETIQUETA_PRONTA	THEN
		passo_ETIQUETA			:=	1003;
	END_IF*)
	
	IF NOT sens_ETIQUETADORA AND NOT GVL_PESAGEM.bit_PESAGEM_ATUAL THEN
		
		tmr_ETIQUETA.IN		:=	TRUE;
		
	END_IF
	
	IF tmr_ETIQUETA.Q	THEN
		tmr_ETIQUETA.IN						:=	FALSE;
		LA_GERAL.do_SAIDA_COLAR_EQUIQUETA	:=	FALSE;
		passo_ETIQUETA		:=	999;
	END_IF
	
//--------------------------------------------------------------------------------------------------------------------------------------------------------------------------------
1003://decide qual o tipo de etiqueta que vai imprimir

	IF GVL_PESAGEM.array_ETIQUETA.1	THEN
		bit_IMPRIMIR_ETIQUETA_1	:=	TRUE;
	ELSE
		bit_IMPRIMIR_ETIQUETA_2	:=	TRUE;
	END_IF
	
	passo_ETIQUETA			:=	1004;
	
	
//--------------------------------------------------------------------------------------------------------------------------------------------------------------------------------
1004://aguarda status de impressão

	IF bit_ETIQUETA_IMPRIMINDO	THEN
		passo_ETIQUETA			:=	1005;
	END_IF
	
//--------------------------------------------------------------------------------------------------------------------------------------------------------------------------------
1005://aguarda confirmação de impressão e liga esteiras

	IF bit_ETIQUETA_CONCLUIDO AND NOT sens_PRODUTO_MERGER	THEN
		GVL_PESAGEM.est_TRANSPORTADOR_ESTAGIO_1	:=	TRUE;
		GVL_PESAGEM.est_TRANNSPORTADOR_MERGER	:=	TRUE;
		passo_ETIQUETA			:=	1006;
	END_IF
	
//--------------------------------------------------------------------------------------------------------------------------------------------------------------------------------
1006://espera pilha de sacolas sair do sensor para reiniciar ciclo

	IF NOT sens_ETIQUETADORA THEN
		passo_ETIQUETA			:=	999;
	END_IF


END_CASE




tmr_PARAR_ESTEIRA(PT:= T#1.8S );
tmr_ETIQUETA(PT:= T#300MS );

END_PROGRAM

// D_PESAGEM/D02_SELEC_ETIQUETA
PROGRAM D02_SELEC_ETIQUETA
VAR
	 fbMarkem : FB_Markem_SelecionarMacro;

    xSelecionarPrograma : BOOL;
    sProgramaMarkem : STRING(24) := '40x50';
	
	bit_LIGA_SCAN	: BOOL;
	
	tmr_1	: TON;
	tmr_2	: TON;
	tmr_3	: TON;
	
	passo_SELEC_ETIQUETA : INT 	:= 9;
	FIRST_SCAN			 : BOOL	:= TRUE;
	teste: BOOL;
END_VAR

	IF	LA_IHM.bit_bt_RESET_PESAGEM	THEN
		passo_SELEC_ETIQUETA	:=	9;
	END_IF

CASE passo_SELEC_ETIQUETA OF

//--------------------------------------------------------------------------------------------------------------------------------------------------------------------------------
9:	

	bit_LIGA_SCAN			:=	FALSE;
	tmr_1.IN				:=	FALSE;
	tmr_2.IN				:=	FALSE;
	tmr_3.IN				:=	FALSE;
	xSelecionarPrograma		:=	FALSE;
	passo_SELEC_ETIQUETA	:=	10;

	
//--------------------------------------------------------------------------------------------------------------------------------------------------------------------------------
10:

	bit_LIGA_SCAN			:=	TRUE;
	IF fbMarkem.xConnected THEN
		passo_SELEC_ETIQUETA	:=	999;
	END_IF
	
//--------------------------------------------------------------------------------------------------------------------------------------------------------------------------------
999:

	IF LA_IHM.bt_DOWNLOAD_RECEITA OR FIRST_SCAN THEN
		tmr_1.IN				:=	TRUE;
		FIRST_SCAN				:=	FALSE;
		passo_SELEC_ETIQUETA	:=	1000;
	END_IF
	
//--------------------------------------------------------------------------------------------------------------------------------------------------------------------------------
1000:

	IF tmr_1.Q	THEN
		tmr_1.IN				:=	FALSE;
		xSelecionarPrograma		:=	TRUE;
		tmr_2.IN				:=	TRUE;
		passo_SELEC_ETIQUETA	:=	1001;
	END_IF
	
//--------------------------------------------------------------------------------------------------------------------------------------------------------------------------------
1001:

	xSelecionarPrograma		:=	FALSE;
	
	IF tmr_2.Q	THEN
		tmr_2.IN				:=	FALSE;
		tmr_3.IN				:=	TRUE;
		xSelecionarPrograma		:=	TRUE;
		passo_SELEC_ETIQUETA	:=	1002;
	END_IF
	
//--------------------------------------------------------------------------------------------------------------------------------------------------------------------------------
1002:

	IF tmr_3.Q	THEN
		tmr_3.IN				:=	FALSE;
		xSelecionarPrograma		:=	FALSE;
		passo_SELEC_ETIQUETA	:=	999;
	END_IF

END_CASE


fbMarkem(
    xEnable     := bit_LIGA_SCAN,
    xSelecionar := xSelecionarPrograma,
    sNomeMacro  := sProgramaMarkem
);

sProgramaMarkem := pvar.rec_ATUAL.NOME;

tmr_1(PT:= T#1500MS);
tmr_2(PT:= T#100MS);
tmr_3(PT:= T#100MS);

END_PROGRAM

// D_PESAGEM/D03_ENTRADAS_REMOTAS
PROGRAM D03_ENTRADAS_REMOTAS
VAR
END_VAR

END_PROGRAM

// D_PESAGEM/D04_SAIDAS_REMOTAS
PROGRAM D04_SAIDAS_REMOTAS
VAR
END_VAR

END_PROGRAM

// LADO_A/01 - LA_GERAL/A00_ENTRADAS
PROGRAM A00_ENTRADAS
VAR
END_VAR


//	SLOT 1		============//============//============//============//============//============//============

	LA_GERAL.di_BT_CMD1_START				:= di_LOCAL_SLOT1_0;
	
	LA_GERAL.di_BT_CMD1_STOP				:= di_LOCAL_SLOT1_1;
	
	LA_GERAL.di_BT_CMD1_RESET				:= di_LOCAL_SLOT1_2;
	
	LA_GERAL.di_BT_CMD2_START				:= di_LOCAL_SLOT1_3;
	
	LA_GERAL.di_BT_CMD2_STOP				:= di_LOCAL_SLOT1_4;
	
	LA_GERAL.di_BT_CMD2_RESET				:= di_LOCAL_SLOT1_5;
	
	//RESERVA								:= di_LOCAL_SLOT1_6;
	
	//RESERVA								:= di_LOCAL_SLOT1_7;
	
	//RESERVA								:= di_LOCAL_SLOT1_8;
	
	LA_GERAL.di_SEG_GERAL_ATIVA				:= di_LOCAL_SLOT1_9;
	
	LA_GERAL.di_SEG_INTERNA_ATIVA			:= di_LOCAL_SLOT1_10;
	
	//RESERVA								:= di_LOCAL_SLOT1_11;
	
	LA_GERAL.di_SEG_PORTA_2					:= di_LOCAL_SLOT1_12;
	
	LA_GERAL.di_SEG_PORTA_1					:= di_LOCAL_SLOT1_13;
	
	//RESERVA								:= di_LOCAL_SLOT1_14;
	
	//RESERVA								:= di_LOCAL_SLOT1_15;
	
	
//	SLOT 2		============//============//============//============//============//============//============

	LA_GERAL.di_ENV_SENS_ATU_GARRA_LD_RC	:= di_LOCAL_SLOT2_0;
	
	LA_GERAL.di_ENV_SENS_ATU_GARRA_LE_RC	:= di_LOCAL_SLOT2_1;
	
	LA_GERAL.di_ENV_SENS_ATU_ABERTURA_AV	:= di_LOCAL_SLOT2_2;
	
	LA_GERAL.di_ENV_SENS_ATU_ABERTURA_RC	:= di_LOCAL_SLOT2_3;
	
	//RESERVA								:= di_LOCAL_SLOT2_4;
	
	//RESERVA								:= di_LOCAL_SLOT2_5;
	
	//RESERVA								:= di_LOCAL_SLOT2_6;
	
	//RESERVA								:= di_LOCAL_SLOT2_7;
	
	//RESERVA								:= di_LOCAL_SLOT2_8;
	
	//RESERVA								:= di_LOCAL_SLOT2_9;
		
	//RESERVA								:= di_LOCAL_SLOT2_10;
	
	//RESERVA								:= di_LOCAL_SLOT2_11;
	
	//RESERVA								:= di_LOCAL_SLOT2_12;
	
	//RESERVA								:= di_LOCAL_SLOT2_13;
	
	//RESERVA								:= di_LOCAL_SLOT2_14;
	
	//RESERVA								:= di_LOCAL_SLOT2_15;

END_PROGRAM

// LADO_A/01 - LA_GERAL/A00_SAIDAS
PROGRAM A00_SAIDAS
VAR
END_VAR

//	SLOT 3		============//============//============//============//============//============//============
	
	do_LOCAL_SLOT3_0	:= LA_GERAL.do_TL1_VERDE;
	
	do_LOCAL_SLOT3_1	:= LA_GERAL.do_TL1_VERMELHO;
	
	do_LOCAL_SLOT3_2	:= LA_GERAL.do_TL1_AMARELO;
	
	do_LOCAL_SLOT3_3	:= LA_GERAL.do_TL2_VERDE;
	
	do_LOCAL_SLOT3_4	:= LA_GERAL.do_TL2_VERMELHO;
	
	do_LOCAL_SLOT3_5	:= LA_GERAL.do_TL2_AMARELO;
	
	do_LOCAL_SLOT3_6	:= LA_GERAL.do_TL1_SONORO;
	
	do_LOCAL_SLOT3_7	:= LA_GERAL.do_SAIDA_COLAR_EQUIQUETA;
	
	
//	SLOT 4		============//============//============//============//============//============//============

	//do_LOCAL_SLOT4_0	:= RESERVA;
	
	//do_LOCAL_SLOT4_1	:= RESERVA;
	
	//do_LOCAL_SLOT4_2	:= RESERVA;
	
	//do_LOCAL_SLOT4_3	:= RESERVA;
	
	do_LOCAL_SLOT4_4	:= LA_GERAL.do_ENV_CORTE_FILME;
	
	//do_LOCAL_SLOT4_5	:= RESERVA;
	
	//do_LOCAL_SLOT4_6	:= RESERVA;
	
	//do_LOCAL_SLOT4_7	:= RESERVA;
	
	
//	SLOT 5		============//============//============//============//============//============//============

	//do_LOCAL_SLOT5_0	:= RESERVA;
	
	//do_LOCAL_SLOT5_1	:= RESERVA;
	
	do_LOCAL_SLOT5_2	:= LA_GERAL.do_ENV_ATU_GARRAS;
	
	do_LOCAL_SLOT5_3	:= LA_GERAL.do_ENV_ATU_ABERTURA;
	
	//do_LOCAL_SLOT5_4	:= RESERVA;
	
	//do_LOCAL_SLOT5_5	:= RESERVA;
	
	//do_LOCAL_SLOT5_6	:= RESERVA;
	
	//do_LOCAL_SLOT5_7	:= RESERVA;

END_PROGRAM

// LADO_A/01 - LA_GERAL/A01_COMANDOS
PROGRAM A01_COMANDOS
VAR
	tmr_AUTO_HABILITAR_EIXOS	: TON;
	tmr_RESET_GERAL				: TON;
	tmr_MAQUINA_ESTAVEL			: TON;
	tmr_MAQUINA_OCIOSA			: TON;
	MICRO_FALHA					: BOOL;
END_VAR

//SAFETY
	IF	NOT LA_GERAL.di_SEG_GERAL_ATIVA 	AND 
		NOT LA_GERAL.di_SEG_INTERNA_ATIVA	THEN
				LA_GERAL.bit_SAFETY_ATIVO			:= TRUE;
	ELSE
				LA_GERAL.bit_SAFETY_ATIVO			:= FALSE;
	END_IF


//LIGAR CELULA
	IF	(LA_GERAL.di_BT_CMD1_START OR LA_GERAL.di_BT_CMD2_START)	AND
		LA_GERAL.bit_SAFETY_ATIVO						THEN
			LA_GERAL.bit_MAQUINA_PRONTA			:= TRUE;
	END_IF
	
	
//DESLIGAR CELULA
	LA_GERAL.bit_BT_DESLIGA	:= LA_GERAL.di_BT_CMD1_STOP OR LA_GERAL.di_BT_CMD2_STOP;

	IF LA_GERAL.bit_BT_DESLIGA OR NOT	LA_GERAL.bit_SAFETY_ATIVO	THEN
			LA_GERAL.bit_MAQUINA_PRONTA			:= FALSE;
	END_IF
	
	
//RESETAR CELULA
	IF 	(LA_GERAL.di_BT_CMD1_RESET OR LA_GERAL.di_BT_CMD2_RESET)	AND
		NOT LA_GERAL.bit_MAQUINA_PRONTA					THEN
		LA_GERAL.bit_SERVOS_RESET	 			:= TRUE;
	ELSE
		LA_GERAL.bit_SERVOS_RESET 				:= FALSE;
	END_IF
	
	
//RESET BITS DE EIXOS DA CELULA	
	IF	LA_GERAL.bit_SERVOS_RESET			THEN
			M0_LA_EMP_X.bit_FAZER_HOME		:= FALSE;
			M1_LA_EMP_GARRA.bit_FAZER_HOME			:= FALSE;
			M2_LA_EMP_GIRO.bit_FAZER_HOME				:= FALSE;
			M3_LA_ENV_Z.bit_FAZER_HOME		:= FALSE;
			M4_LA_ENV_X.bit_FAZER_HOME		:= FALSE;
			M5_LA_ENV_GIRO_LD.bit_FAZER_HOME		:= FALSE;
			M6_LA_ENV_GIRO_LE.bit_FAZER_HOME		:= FALSE;
		
			LA_EMP.bit_EIXO_X_EMPILHADOR_MOVER_ABS 	 		:= FALSE;
			LA_EMP.bit_EIXO_GARRA_EMPILHADOR_MOVER_ABS 		:= FALSE;
			LA_EMP.bit_EIXO_GIRO_MESA_MOVER_ABS 			:= FALSE;
			LA_ENV.bit_EIXO_Z_ENVOLVEDOR_MOVER_ABS 			:= FALSE;
			LA_ENV.bit_EIXO_X_ENVOLVEDOR_MOVER_ABS 			:= FALSE;
			LA_ENV.bit_EIXO_GIRO_ENVOLVEDOR_LD_MOVER_ABS 	:= FALSE;
			LA_ENV.bit_EIXO_GIRO_ENVOLVEDOR_LE_MOVER_ABS 	:= FALSE;
			
			LA_EMP.bit_EIXO_X_EMPILHADOR_MOVER_REL 	 		:= FALSE;
			LA_EMP.bit_EIXO_GARRA_EMPILHADOR_MOVER_REL 		:= FALSE;
			LA_EMP.bit_EIXO_GIRO_MESA_MOVER_REL 			:= FALSE;
			LA_ENV.bit_EIXO_Z_ENVOLVEDOR_MOVER_REL 			:= FALSE;
			LA_ENV.bit_EIXO_X_ENVOLVEDOR_MOVER_REL 			:= FALSE;
			LA_ENV.bit_EIXO_GIRO_ENVOLVEDOR_LD_MOVER_REL 	:= FALSE;
			LA_ENV.bit_EIXO_GIRO_ENVOLVEDOR_LE_MOVER_REL 	:= FALSE;
			
	END_IF
	
	IF LA_GERAL.bit_SERVOS_RESET OR LA_GERAL.TESTE_Z THEN
		LA_GERAL.RESET_Z	:=	TRUE;
	ELSE
		LA_GERAL.RESET_Z	:=	FALSE;
	END_IF
	
//SE TODOS OS CONJUNTOS RESETAREM, COMEÇA A RODAR CELULA
	IF	LA_GERAL.bit_MAQUINA_PRONTA						AND
		LA_IHM.bit_EIXO_X_EMPILHADOR_HABILITADO			AND
		LA_IHM.bit_EIXO_GARRA_EMPILHADOR_HABILITADO				AND
		LA_IHM.bit_EIXO_GIRO_MESA_HABILITADO					(*AND
		M03_DRV_EIXO_Z_ENVOLVEDOR.bit_HABILITADO			AND
		M04_DRV_EIXO_X_ENVOLVEDOR.bit_HABILITADO			AND
		M05_DRV_GIRO_ENVOLVEDOR_LD.bit_HABILITADO			AND
		M06_DRV_GIRO_ENVOLVEDOR_LE.bit_HABILITADO*)			THEN
			LA_GERAL.bit_MAQUINA_RODANDO	:= TRUE;
			LA_IHM.bit_MAQUINA_MANUAL		:= FALSE;
	ELSE
			LA_GERAL.bit_MAQUINA_RODANDO	:= FALSE;
	END_IF
	
	
// RESET GERAL
	tmr_RESET_GERAL (PT := T#2000MS);
	
	tmr_RESET_GERAL.IN := 	LA_GERAL.di_BT_CMD1_RESET OR LA_GERAL.di_BT_CMD2_RESET;
	
	IF	tmr_RESET_GERAL.Q	THEN
			LA_GERAL.bit_RESET_GERAL := TRUE;	
	END_IF
	
//EIXOS
	IF	LA_GERAL.bit_AUTO_HABILITAR_EIXOS		OR
		LA_IHM.bit_MANUAL_HABILITAR_EIXOS		THEN
			LA_GERAL.bit_HABILITAR_EIXOS	:= TRUE;
	ELSE
			LA_GERAL.bit_HABILITAR_EIXOS	:= FALSE;
	END_IF
	
	IF	NOT LA_GERAL.bit_MAQUINA_MANUAL	THEN
				LA_IHM.bit_MANUAL_HABILITAR_EIXOS	:= FALSE;
	END_IF
	
	IF	LA_GERAL.bit_SAFETY_ATIVO AND (LA_GERAL.di_BT_CMD1_RESET OR LA_GERAL.di_BT_CMD2_RESET)	THEN
			LA_GERAL.bit_AUTO_HABILITAR_EIXOS	:= TRUE;
	END_IF
	
	
	IF NOT	LA_GERAL.bit_SAFETY_ATIVO		THEN
			LA_GERAL.bit_AUTO_HABILITAR_EIXOS	:= FALSE;
	END_IF
	
//tmr_AUTO_HABILITAR_EIXOS (IN:= NOT GVL_CELULA.bit_SAFETY_ATIVO, PT:= T#10S);

	IF 	LA_GERAL.bit_EIXO_X_EMPILHADOR_PRONTO			AND
		LA_GERAL.bit_EIXO_GARRA_EMPILHADOR_PRONTO		AND
		LA_GERAL.bit_EIXO_GIRO_MESA_PRONTO			AND
		LA_GERAL.bit_EIXO_Z_ENVOLVEDOR_PRONTO			AND
		LA_GERAL.bit_EIXO_X_ENVOLVEDOR_PRONTO			AND
		LA_GERAL.bit_EIXO_GIRO_ENVOLVEDOR_LD_PRONTO	AND
		LA_GERAL.bit_EIXO_GIRO_ENVOLVEDOR_LD_PRONTO	THEN
			LA_GERAL.bit_EIXOS_PRONTOS	:=	TRUE;
	ELSE
			LA_GERAL.bit_EIXOS_PRONTOS	:=	FALSE;
		
	END_IF

//LIGAR ESTEIRAS
	
	//ESTEIRAS EMPILHADOR
	IF	LA_GERAL.bit_SAFETY_ATIVO AND (LA_EMP.est_INSPECAO_EMPILHADOR OR LA_IHM.est_INSPECAO_EMPILHADOR) THEN
			SPEED_A_EST_INSPECAO	:=	TRUE;
			SPEED_B_EST_INSPECAO	:=	TRUE;
	ELSE
			SPEED_A_EST_INSPECAO	:=	FALSE;
			SPEED_B_EST_INSPECAO	:=	FALSE;
	END_IF
	
	IF LA_GERAL.bit_SAFETY_ATIVO AND	(LA_EMP.est_ROLETES_GIRO_MESA OR LA_IHM.est_ROLETES_GIRO_MESA) THEN
			SPEED_A_MESA_GIRO	:=	TRUE;
			SPEED_B_MESA_GIRO	:=	TRUE;
	ELSE
			SPEED_A_MESA_GIRO	:=	FALSE;
			SPEED_B_MESA_GIRO	:=	FALSE;
	END_IF
//--------------------------////--------------------------////--------------------------////--------------------------////--------------------------//	
	//ESTEIRAS ENVOLVEDOR
	IF LA_GERAL.bit_SAFETY_ATIVO AND	((LA_ENV.est_ENTRADA_ENVOLVEDOR AND NOT LA_IHM.bit_MAQUINA_MANUAL) OR LA_IHM.est_ENVOLVEDOR_ENTRADA) THEN
			SPEED_A_ENTRADA_ENVOLVEDOR	:=	TRUE;
	ELSE
			SPEED_A_ENTRADA_ENVOLVEDOR	:=	FALSE;
	END_IF
	
	IF LA_GERAL.bit_SAFETY_ATIVO AND	((LA_ENV.est_TRANSPORTADOR_ENVOLVEDOR AND NOT LA_IHM.bit_MAQUINA_MANUAL) OR LA_IHM.est_TRANSPORTADOR_ENVOLVEDOR) THEN
			eest_TRANS_ENVOLVEDOR_DI2	:=	TRUE;
	ELSE
			eest_TRANS_ENVOLVEDOR_DI2	:=	FALSE;
	END_IF
	
	IF LA_GERAL.bit_SAFETY_ATIVO AND	(LA_ENV.est_SAIDA_ENVOLVEDOR OR LA_IHM.est_ENVOLVEDOR_SAIDA) THEN
			SPEED_A_TRANSP_SAIDA_1	:=	TRUE;
	ELSE
			SPEED_A_TRANSP_SAIDA_1	:=	FALSE;
	END_IF
//--------------------------////--------------------------////--------------------------////--------------------------////--------------------------//	
	//ESTEIRAS PESAGEM DE PRODUTO
	IF LA_GERAL.bit_SAFETY_ATIVO AND (GVL_PESAGEM.est_MESA_DE_TRANSFERENCIA OR LA_IHM.est_MESA_DE_TRANSFERENCIA) AND (NOT GVL_PESAGEM.est_MESA_DE_TRANSFERENCIA_REVERSE AND NOT LA_IHM.est_MESA_DE_TRANSFERENCIA_REVERSE) THEN
			est_MESA_TRANS_PESAGEM_DI1 := TRUE;
			est_MESA_TRANS_PESAGEM_DI3 := FALSE;
	ELSE
			est_MESA_TRANS_PESAGEM_DI1 := FALSE;
	END_IF
	
	IF LA_GERAL.bit_SAFETY_ATIVO AND (GVL_PESAGEM.est_REJEITO_PRODUTO OR LA_IHM.est_REJEITO_PRODUTO) THEN
			SPEED_A_REJEITO_PRODUTO := TRUE;
	ELSE
			SPEED_A_REJEITO_PRODUTO := FALSE;
	END_IF
	
	IF LA_GERAL.bit_SAFETY_ATIVO AND (GVL_PESAGEM.est_TRANSPORTADOR_PESAGEM OR LA_IHM.est_TRANSPORTADOR_PESAGEM) THEN
			SPEED_A_MESA_TRANSFER	:=	TRUE;
			//SPEED_B_MESA_TRANSFER	:=	TRUE;
	ELSE
			SPEED_A_MESA_TRANSFER	:=	FALSE;
			SPEED_B_MESA_TRANSFER	:=	FALSE;
	END_IF
	
	IF LA_GERAL.bit_SAFETY_ATIVO AND (GVL_PESAGEM.est_TRANSPORTADOR_ESTAGIO_1 OR LA_IHM.est_TRANSPORTADOR_ESTAGIO_1) THEN
			SPEED_A_ESTAGIO_1 := TRUE;
	ELSE
			SPEED_A_ESTAGIO_1 := FALSE;
	END_IF
	
//--------------------------////--------------------------////--------------------------////--------------------------////--------------------------//
	//INVERSÃO DE ETEIRAS
	IF LA_GERAL.bit_SAFETY_ATIVO AND (LA_EMP.est_INSPECAO_EMPILHADOR_REVERSE OR LA_IHM.est_INSPECAO_EMPILHADOR_REVERSE) THEN
			REVERSE_EST_INSPECAO := TRUE;
	ELSE
			REVERSE_EST_INSPECAO := FALSE;
	END_IF
	
	IF LA_GERAL.bit_SAFETY_ATIVO AND (LA_EMP.est_ROLETES_GIRO_MESA_REVERSE OR LA_IHM.est_ROLETES_GIRO_MESA_REVERSE) THEN
			REVERSE_MESA_GIRO := TRUE;
	ELSE
			REVERSE_MESA_GIRO := FALSE;
	END_IF

	IF  (GVL_PESAGEM.est_MESA_DE_TRANSFERENCIA OR LA_IHM.est_MESA_DE_TRANSFERENCIA) 				AND
		(GVL_PESAGEM.est_MESA_DE_TRANSFERENCIA_REVERSE OR LA_IHM.est_MESA_DE_TRANSFERENCIA_REVERSE)AND
		LA_GERAL.bit_SAFETY_ATIVO			 														THEN
			est_MESA_TRANS_PESAGEM_DI3 := TRUE;
			est_MESA_TRANS_PESAGEM_DI1 := FALSE;
	ELSE
			est_MESA_TRANS_PESAGEM_DI3 := FALSE;
	END_IF
	
	IF LA_GERAL.bit_SAFETY_ATIVO AND (GVL_PESAGEM.est_TRANSPORTADOR_PESAGEM_REVERSE OR LA_IHM.est_TRANSPORTADOR_PESAGEM_REVERSE) THEN
			REVERSE_MESA_TRANSFER := TRUE;
	ELSE
			REVERSE_MESA_TRANSFER := FALSE;
	END_IF
//--------------------------////--------------------------////--------------------------////--------------------------////--------------------------//
	
//BIT MAQUINA ESTAVEL 
	tmr_MAQUINA_ESTAVEL	(IN:= LA_GERAL.bit_MAQUINA_RODANDO, PT := T#5000MS);
	LA_GERAL.bit_MAQUINA_ESTAVEL	:= tmr_MAQUINA_ESTAVEL.Q;


//---------------------//---------------------------------------------//---------------------------------------------//------------------------
//---------------------//------------------------STATUS MAQUINA---------------------//------------------------


//STATUS MAQUINA RODANDO
	IF 	LA_GERAL.bit_MAQUINA_RODANDO 			AND 
	NOT LA_GERAL.bit_STATUS_PARADA 			THEN
		 LA_GERAL.bit_STATUS_RODANDO	:=	TRUE;
	ELSE
		 LA_GERAL.bit_STATUS_RODANDO	:=	FALSE;
	END_IF
	
//STATUS MAQUINA PARADA
	IF 	NOT LA_GERAL.bit_SAFETY_ATIVO 	 	THEN
		 	LA_GERAL.bit_STATUS_PARADA		:=	TRUE;
	ELSE
			LA_GERAL.bit_STATUS_PARADA		:=	FALSE;
	END_IF
	
//STATUS MAQUINA OCIOSA
	IF  LA_GERAL.bit_SAFETY_ATIVO 				AND
		LA_GERAL.bit_MAQUINA_RODANDO				AND
	NOT LA_GERAL.bit_EIXO_GERAL_MOVENDO 			THEN
		 tmr_MAQUINA_OCIOSA.IN			:=	TRUE;
	ELSE
		tmr_MAQUINA_OCIOSA.IN			:=	FALSE;
	END_IF
	
	IF tmr_MAQUINA_OCIOSA.Q OR	(NOT LA_GERAL.bit_MAQUINA_RODANDO AND LA_GERAL.bit_SAFETY_ATIVO) THEN
		LA_GERAL.bit_STATUS_OCIOSA	:=	TRUE;
	ELSE
		LA_GERAL.bit_STATUS_OCIOSA	:=	FALSE;
	END_IF
	
	
LA_IHM.bit_PORTA_1		:= LA_GERAL.di_SEG_PORTA_1;
LA_IHM.bit_PORTA_2 		:= LA_GERAL.di_SEG_PORTA_2;
	
//TIMERS		
	tmr_MAQUINA_OCIOSA (PT:= T#15S);

END_PROGRAM

// LADO_A/04 - LA_MOTION/M0_LA_EMP_X
PROGRAM M0_LA_EMP_X
VAR
	fb_POWER				: MC_Power;
	fb_RESET				: MC_Reset;
	fb_LER_POS_ATUAL		: MC_ReadActualPosition;
	fb_HOME					: MC_Home;
	fb_MOVER_ABS			: MC_MoveAbsolute;
	fb_MOVER_REL			: MC_MoveRelative;
	fb_MOVER_JOG			: MC_JOG;
	fb_MOVER_STOP			: MC_STOP;

	bit_POWER_ERRO			: BOOL;
	bit_HOME_ERRO			: BOOL;
	bit_MOVE_ABS_ERRO		: BOOL;
	bit_MOVE_REL_ERRO		: BOOL;
	bit_MOVE_JOG_ERRO		: BOOL;
	
	bit_HABILITADO			: BOOL;
	bit_HOME_FEITO			: BOOL;
	bit_HOME_FAZENDO		: BOOL;
	bit_MOVE_ABS_FEITO		: BOOL;
	bit_MOVE_ABS_FAZENDO	: BOOL;
	bit_MOVE_REL_FEITO		: BOOL;
	bit_MOVE_REL_FAZENDO	: BOOL;
	bit_HABILITAR_EIXOS		: BOOL;
	bit_EIXO_DRV_MOVER_ABS	: BOOL;
	bit_DRV_JOG_FORWARD		: BOOL;
	bit_DRV_JOG_REVERSE		: BOOL;
	bit_DRV_JOG_STOP		: BOOL;
	bit_SERVOS_RESET		: BOOL;
	info_MOTOR_PASSO_POS_ATUAL: LREAL;
END_VAR


VAR_INPUT
	
	ABS_MOVER				: EIXO_MOVER;
	REL_MOVER				: EIXO_MOVER;
	
	bit_FAZER_HOME			: BOOL;
END_VAR

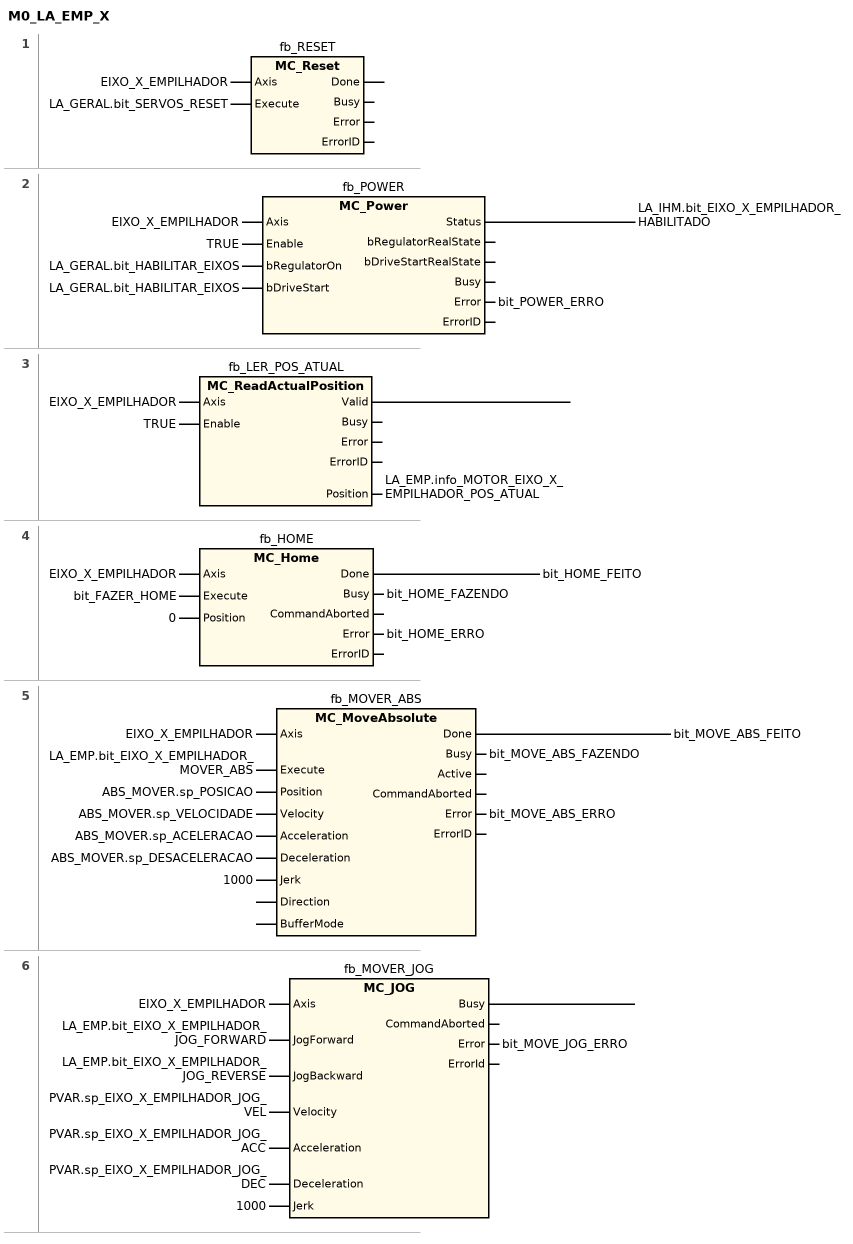
// NETWORK 1
fb_RESET(Axis := EIXO_X_EMPILHADOR, Execute := LA_GERAL.bit_SERVOS_RESET); // MC_Reset

// NETWORK 2
fb_POWER(
    Axis := EIXO_X_EMPILHADOR,
    Enable := TRUE,
    bRegulatorOn := LA_GERAL.bit_HABILITAR_EIXOS,
    bDriveStart := LA_GERAL.bit_HABILITAR_EIXOS,
    Error => bit_POWER_ERRO); // MC_Power
LA_IHM.bit_EIXO_X_EMPILHADOR_HABILITADO := fb_POWER.Status;

// NETWORK 3
fb_LER_POS_ATUAL(
    Axis := EIXO_X_EMPILHADOR,
    Enable := TRUE,
    Position => LA_EMP.info_MOTOR_EIXO_X_EMPILHADOR_POS_ATUAL); // MC_ReadActualPosition

// NETWORK 4
fb_HOME(
    Axis := EIXO_X_EMPILHADOR,
    Execute := bit_FAZER_HOME,
    Position := 0,
    Busy => bit_HOME_FAZENDO,
    Error => bit_HOME_ERRO); // MC_Home
bit_HOME_FEITO := fb_HOME.Done;

// NETWORK 5
fb_MOVER_ABS(
    Axis := EIXO_X_EMPILHADOR,
    Execute := LA_EMP.bit_EIXO_X_EMPILHADOR_MOVER_ABS,
    Position := ABS_MOVER.sp_POSICAO,
    Velocity := ABS_MOVER.sp_VELOCIDADE,
    Acceleration := ABS_MOVER.sp_ACELERACAO,
    Deceleration := ABS_MOVER.sp_DESACELERACAO,
    Jerk := 1000,
    Busy => bit_MOVE_ABS_FAZENDO,
    Error => bit_MOVE_ABS_ERRO); // MC_MoveAbsolute
bit_MOVE_ABS_FEITO := fb_MOVER_ABS.Done;

// NETWORK 6
fb_MOVER_JOG(
    Axis := EIXO_X_EMPILHADOR,
    JogForward := LA_EMP.bit_EIXO_X_EMPILHADOR_JOG_FORWARD,
    JogBackward := LA_EMP.bit_EIXO_X_EMPILHADOR_JOG_REVERSE,
    Velocity := PVAR.sp_EIXO_X_EMPILHADOR_JOG_VEL,
    Acceleration := PVAR.sp_EIXO_X_EMPILHADOR_JOG_ACC,
    Deceleration := PVAR.sp_EIXO_X_EMPILHADOR_JOG_DEC,
    Jerk := 1000,
    Error => bit_MOVE_JOG_ERRO); // MC_JOG

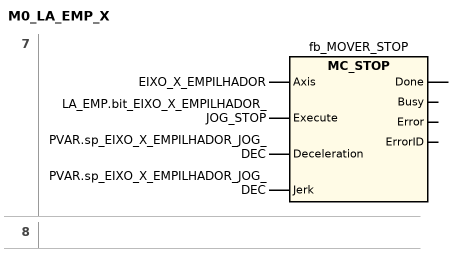
// NETWORK 7
fb_MOVER_STOP(
    Axis := EIXO_X_EMPILHADOR,
    Execute := LA_EMP.bit_EIXO_X_EMPILHADOR_JOG_STOP,
    Deceleration := PVAR.sp_EIXO_X_EMPILHADOR_JOG_DEC,
    Jerk := PVAR.sp_EIXO_X_EMPILHADOR_JOG_DEC); // MC_STOP

// NETWORK 8

END_PROGRAM

// LADO_A/04 - LA_MOTION/M1_LA_EMP_GARRA
PROGRAM M1_LA_EMP_GARRA
VAR
	fb_POWER				: MC_Power;
	fb_RESET				: MC_Reset;
	fb_LER_POS_ATUAL		: MC_ReadActualPosition;
	fb_HOME					: MC_Home;
	fb_MOVER_ABS			: MC_MoveAbsolute;
	fb_MOVER_REL			: MC_MoveRelative;
	fb_MOVER_JOG			: MC_JOG;
	fb_MOVER_STOP			: MC_STOP;

	bit_POWER_ERRO			: BOOL;
	bit_HOME_ERRO			: BOOL;
	bit_MOVE_ABS_ERRO		: BOOL;
	bit_MOVE_REL_ERRO		: BOOL;
	bit_MOVE_JOG_ERRO		: BOOL;
	
	bit_HABILITADO			: BOOL;
	bit_HOME_FEITO			: BOOL;
	bit_HOME_FAZENDO		: BOOL;
	bit_MOVE_ABS_FEITO		: BOOL;
	bit_MOVE_ABS_FAZENDO	: BOOL;
	bit_MOVE_REL_FEITO		: BOOL;
	bit_MOVE_REL_FAZENDO	: BOOL;
	bit_HABILITAR_EIXOS		: BOOL;
	bit_EIXO_DRV_MOVER_ABS	: BOOL;
	bit_DRV_JOG_FORWARD		: BOOL;
	bit_DRV_JOG_REVERSE		: BOOL;
	bit_DRV_JOG_STOP		: BOOL;
	bit_SERVOS_RESET		: BOOL;
	info_MOTOR_PASSO_POS_ATUAL: LREAL;
END_VAR


VAR_INPUT
	
	ABS_MOVER				: EIXO_MOVER;
	REL_MOVER				: EIXO_MOVER;
	
